LIN {X 0,Y 675.561,Z 368.02,A -85,B 0,C 180,E1 -4011.807,E2 -4011.807} C_VEL
LIN {X 0,Y 675.363,Z 376.661,A -85,B 0,C 180,E1 -4012.443,E2 -4012.443} C_VEL
LIN {X 0,Y 680.703,Z 399.355,A -85,B 0,C 180,E1 -4013.079,E2 -4013.079} C_VEL
LIN {X 0,Y 678.008,Z 663.117,A -85,B 0,C 180,E1 -4016.26,E2 -4016.26} C_VEL
LIN {X 0,Y 676.914,Z 767.818,A -85,B 0,C 180,E1 -4017.526,E2 -4017.526} C_VEL
LIN {X 0,Y 676.255,Z 793.274,A -85,B 0,C 180,E1 -4017.987,E2 -4017.987} C_VEL
LIN {X 0,Y 675.528,Z 814.444,A -85,B 0,C 180,E1 -4018.503,E2 -4018.503} C_VEL
LIN {X 0,Y 674.622,Z 838.547,A -85,B 0,C 180,E1 -4019.247,E2 -4019.247} C_VEL
LIN {X 0,Y 673.655,Z 859.342,A -85,B 0,C 180,E1 -4020.036,E2 -4020.036} C_VEL
LIN {X 0,Y 672.656,Z 880.17,A -85,B 0,C 180,E1 -4020.961,E2 -4020.961} C_VEL
LIN {X 0,Y 671.429,Z 902.313,A -85,B 0,C 180,E1 -4022.121,E2 -4022.121} C_VEL
LIN {X 0,Y 670.354,Z 922.188,A -85,B 0,C 180,E1 -4023.323,E2 -4023.323} C_VEL
LIN {X 0,Y 669.167,Z 942.614,A -85,B 0,C 180,E1 -4024.748,E2 -4024.748} C_VEL
LIN {X 0,Y 668.229,Z 959.683,A -85,B 0,C 180,E1 -4026.101,E2 -4026.101} C_VEL
LIN {X 0,Y 667.192,Z 978.606,A -85,B 0,C 180,E1 -4027.811,E2 -4027.811} C_VEL
LIN {X 0,Y 666.433,Z 993.633,A -85,B 0,C 180,E1 -4029.355,E2 -4029.355} C_VEL
LIN {X 0,Y 665.654,Z 1009.818,A -85,B 0,C 180,E1 -4031.249,E2 -4031.249} C_VEL
LIN {X 0,Y 665.145,Z 1022.539,A -85,B 0,C 180,E1 -4032.956,E2 -4032.956} C_VEL
LIN {X 0,Y 664.665,Z 1035.765,A -85,B 0,C 180,E1 -4035.004,E2 -4035.004} C_VEL
LIN {X 0,Y 664.369,Z 1045.92,A -85,B 0,C 180,E1 -4036.844,E2 -4036.844} C_VEL
LIN {X 0,Y 664.133,Z 1055.927,A -85,B 0,C 180,E1 -4039,E2 -4039} C_VEL
LIN {X 0,Y 664.022,Z 1062.817,A -85,B 0,C 180,E1 -4040.815,E2 -4040.815} C_VEL
LIN {X 0,Y 663.962,Z 1069.244,A -85,B 0,C 180,E1 -4042.907,E2 -4042.907} C_VEL
LIN {X 0,Y 663.925,Z 1073.656,A -85,B 0,C 180,E1 -4044.902,E2 -4044.902} C_VEL
LIN {X 0,Y 663.917,Z 1076.574,A -85,B 0,C 180,E1 -4046.806,E2 -4046.806} C_VEL
LIN {X 0,Y 663.91,Z 1078.261,A -85,B 0,C 180,E1 -4049.051,E2 -4049.051} C_VEL
LIN {X 0,Y 663.905,Z 1078.283,A -85,B 0,C 180,E1 -4050.863,E2 -4050.863} C_VEL
LIN {X 0,Y 663.916,Z 1076.799,A -85,B 0,C 180,E1 -4053.022,E2 -4053.022} C_VEL
LIN {X 0,Y 663.925,Z 1073.815,A -85,B 0,C 180,E1 -4055.011,E2 -4055.011} C_VEL
LIN {X 0,Y 663.956,Z 1069.451,A -85,B 0,C 180,E1 -4057.007,E2 -4057.007} C_VEL
LIN {X 0,Y 664.011,Z 1063.119,A -85,B 0,C 180,E1 -4059.097,E2 -4059.097} C_VEL
LIN {X 0,Y 664.128,Z 1056.186,A -85,B 0,C 180,E1 -4060.935,E2 -4060.935} C_VEL
LIN {X 0,Y 664.356,Z 1046.484,A -85,B 0,C 180,E1 -4063.047,E2 -4063.047} C_VEL
LIN {X 0,Y 664.649,Z 1036.288,A -85,B 0,C 180,E1 -4064.907,E2 -4064.907} C_VEL
LIN {X 0,Y 665.121,Z 1023.16,A -85,B 0,C 180,E1 -4066.956,E2 -4066.956} C_VEL
LIN {X 0,Y 665.624,Z 1010.525,A -85,B 0,C 180,E1 -4068.661,E2 -4068.661} C_VEL
LIN {X 0,Y 666.404,Z 994.378,A -85,B 0,C 180,E1 -4070.565,E2 -4070.565} C_VEL
LIN {X 0,Y 667.168,Z 979.013,A -85,B 0,C 180,E1 -4072.149,E2 -4072.149} C_VEL
LIN {X 0,Y 668.189,Z 960.506,A -85,B 0,C 180,E1 -4073.83,E2 -4073.83} C_VEL
LIN {X 0,Y 669.129,Z 943.22,A -85,B 0,C 180,E1 -4075.206,E2 -4075.206} C_VEL
LIN {X 0,Y 670.317,Z 922.909,A -85,B 0,C 180,E1 -4076.631,E2 -4076.631} C_VEL
LIN {X 0,Y 671.389,Z 903.048,A -85,B 0,C 180,E1 -4077.837,E2 -4077.837} C_VEL
LIN {X 0,Y 672.604,Z 881.268,A -85,B 0,C 180,E1 -4078.988,E2 -4078.988} C_VEL
LIN {X 0,Y 673.605,Z 860.476,A -85,B 0,C 180,E1 -4079.918,E2 -4079.918} C_VEL
LIN {X 0,Y 674.538,Z 840.351,A -85,B 0,C 180,E1 -4080.688,E2 -4080.688} C_VEL
LIN {X 0,Y 675.503,Z 815.099,A -85,B 0,C 180,E1 -4081.479,E2 -4081.479} C_VEL
LIN {X 0,Y 676.235,Z 793.801,A -85,B 0,C 180,E1 -4082.002,E2 -4082.002} C_VEL
LIN {X 0,Y 676.909,Z 768.357,A -85,B 0,C 180,E1 -4082.466,E2 -4082.466} C_VEL
LIN {X 0,Y 677.778,Z 687.025,A -85,B 0,C 180,E1 -4083.455,E2 -4083.455} C_VEL
LIN {X 0,Y 680.316,Z 433.987,A -85,B 0,C 180,E1 -4086.5,E2 -4086.5} C_VEL
LIN {X 0,Y 680.519,Z 397.746,A -85,B 0,C 180,E1 -4086.954,E2 -4086.954} C_VEL
LIN {X 0,Y 675.309,Z 375.991,A -85,B 0,C 180,E1 -4087.591,E2 -4087.591} C_VEL
LIN {X 0,Y 675.511,Z 367.275,A -85,B 0,C 180,E1 -4088.256,E2 -4088.256} C_VEL
LIN {X 0,Y 667.62,Z 346.692,A -85,B 0,C 180,E1 -4090.429,E2 -4090.429} C_VEL
LIN {X 0,Y 664.607,Z 338.449,A -85,B 0,C 180,E1 -4091.345,E2 -4091.345} C_VEL
LIN {X 0,Y 664.579,Z 338.447,A -85,B 0,C 180,E1 -4094.035,E2 -4094.035} C_VEL
LIN {X 0,Y 664.647,Z 338.444,A -85,B 0,C 180,E1 -4097.04,E2 -4097.04} C_VEL
LIN {X 0,Y 664.579,Z 338.439,A -85,B 0,C 180,E1 -4099.913,E2 -4099.913} C_VEL
LIN {X 0,Y 664.618,Z 338.438,A -85,B 0,C 180,E1 -4102.678,E2 -4102.678} C_VEL
LIN {X 0,Y 664.591,Z 338.44,A -85,B 0,C 180,E1 -4105.758,E2 -4105.758} C_VEL
LIN {X 0,Y 664.585,Z 338.439,A -85,B 0,C 180,E1 -4108.427,E2 -4108.427} C_VEL
LIN {X 0,Y 664.636,Z 338.439,A -85,B 0,C 180,E1 -4111.471,E2 -4111.471} C_VEL
LIN {X 0,Y 664.579,Z 338.441,A -85,B 0,C 180,E1 -4114.322,E2 -4114.322} C_VEL
LIN {X 0,Y 664.652,Z 338.43,A -85,B 0,C 180,E1 -4117.255,E2 -4117.255} C_VEL
LIN {X 0,Y 664.581,Z 338.436,A -85,B 0,C 180,E1 -4120.213,E2 -4120.213} C_VEL
LIN {X 0,Y 664.62,Z 338.438,A -85,B 0,C 180,E1 -4123.03,E2 -4123.03} C_VEL
LIN {X 0,Y 664.595,Z 338.44,A -85,B 0,C 180,E1 -4126.071,E2 -4126.071} C_VEL
LIN {X 0,Y 664.589,Z 338.44,A -85,B 0,C 180,E1 -4128.809,E2 -4128.809} C_VEL
LIN {X 0,Y 664.617,Z 338.445,A -85,B 0,C 180,E1 -4131.957,E2 -4131.957} C_VEL
LIN {X 0,Y 664.581,Z 338.436,A -85,B 0,C 180,E1 -4134.734,E2 -4134.734} C_VEL
LIN {X 0,Y 664.649,Z 338.44,A -85,B 0,C 180,E1 -4137.758,E2 -4137.758} C_VEL
LIN {X 0,Y 664.58,Z 338.43,A -85,B 0,C 180,E1 -4140.603,E2 -4140.603} C_VEL
LIN {X 0,Y 664.629,Z 338.438,A -85,B 0,C 180,E1 -4143.45,E2 -4143.45} C_VEL
LIN {X 0,Y 664.592,Z 338.438,A -85,B 0,C 180,E1 -4146.479,E2 -4146.479} C_VEL
LIN {X 0,Y 664.593,Z 338.44,A -85,B 0,C 180,E1 -4149.177,E2 -4149.177} C_VEL
LIN {X 0,Y 664.615,Z 338.443,A -85,B 0,C 180,E1 -4152.335,E2 -4152.335} C_VEL
LIN {X 0,Y 664.584,Z 338.437,A -85,B 0,C 180,E1 -4155.087,E2 -4155.087} C_VEL
LIN {X 0,Y 664.65,Z 338.438,A -85,B 0,C 180,E1 -4158.054,E2 -4158.054} C_VEL
LIN {X 0,Y 664.582,Z 338.434,A -85,B 0,C 180,E1 -4160.982,E2 -4160.982} C_VEL
LIN {X 0,Y 664.64,Z 338.439,A -85,B 0,C 180,E1 -4163.872,E2 -4163.872} C_VEL
LIN {X 0,Y 664.589,Z 338.443,A -85,B 0,C 180,E1 -4166.928,E2 -4166.928} C_VEL
LIN {X 0,Y 664.605,Z 338.431,A -85,B 0,C 180,E1 -4169.668,E2 -4169.668} C_VEL
LIN {X 0,Y 664.605,Z 338.436,A -85,B 0,C 180,E1 -4172.794,E2 -4172.794} C_VEL
LIN {X 0,Y 664.589,Z 338.441,A -85,B 0,C 180,E1 -4175.517,E2 -4175.517} C_VEL
LIN {X 0,Y 664.648,Z 338.437,A -85,B 0,C 180,E1 -4176.373,E2 -4176.373} C_VEL
LIN {X 0,Y 663.642,Z 338.561,A -85,B 0,C 180,E1 -4177.037,E2 -4177.037} C_VEL
LIN {X 0,Y 657.183,Z 339.369,A -85,B 0,C 180,E1 -4178.898,E2 -4178.898} C_VEL
LIN {X 0,Y 656.644,Z 339.428,A -85,B 0,C 180,E1 -4179.383,E2 -4179.383} C_VEL
LIN {X 0,Y 656.711,Z 339.428,A -85,B 0,C 180,E1 -4182.298,E2 -4182.298} C_VEL
LIN {X 0,Y 656.647,Z 339.421,A -85,B 0,C 180,E1 -4185.326,E2 -4185.326} C_VEL
LIN {X 0,Y 656.688,Z 339.425,A -85,B 0,C 180,E1 -4188.171,E2 -4188.171} C_VEL
LIN {X 0,Y 656.656,Z 339.438,A -85,B 0,C 180,E1 -4191.257,E2 -4191.257} C_VEL
LIN {X 0,Y 656.715,Z 339.481,A -85,B 0,C 180,E1 -4192.392,E2 -4192.392} C_VEL
LIN {X 0,Y 660.299,Z 349.162,A -85,B 0,C 180,E1 -4193.484,E2 -4193.484} C_VEL
LIN {X 0,Y 672.665,Z 370.1,A -85,B 0,C 180,E1 -4194.601,E2 -4194.601} C_VEL
LIN {X 0,Y 674.3,Z 373.32,A -85,B 0,C 180,E1 -4194.751,E2 -4194.751} C_VEL
LIN {X 0,Y 671.619,Z 610.249,A -85,B 0,C 180,E1 -4197.648,E2 -4197.648} C_VEL
LIN {X 0,Y 670.159,Z 737.628,A -85,B 0,C 180,E1 -4199.2,E2 -4199.2} C_VEL
LIN {X 0,Y 669.456,Z 763.152,A -85,B 0,C 180,E1 -4199.664,E2 -4199.664} C_VEL
LIN {X 0,Y 668.682,Z 784.147,A -85,B 0,C 180,E1 -4200.179,E2 -4200.179} C_VEL
LIN {X 0,Y 667.747,Z 806.973,A -85,B 0,C 180,E1 -4200.879,E2 -4200.879} C_VEL
LIN {X 0,Y 666.641,Z 828.781,A -85,B 0,C 180,E1 -4201.708,E2 -4201.708} C_VEL
LIN {X 0,Y 665.571,Z 849.482,A -85,B 0,C 180,E1 -4202.632,E2 -4202.632} C_VEL
LIN {X 0,Y 664.202,Z 872.164,A -85,B 0,C 180,E1 -4203.827,E2 -4203.827} C_VEL
LIN {X 0,Y 663.039,Z 891.79,A -85,B 0,C 180,E1 -4205.023,E2 -4205.023} C_VEL
LIN {X 0,Y 661.729,Z 912.624,A -85,B 0,C 180,E1 -4206.49,E2 -4206.49} C_VEL
LIN {X 0,Y 660.649,Z 930.299,A -85,B 0,C 180,E1 -4207.907,E2 -4207.907} C_VEL
LIN {X 0,Y 659.548,Z 948.684,A -85,B 0,C 180,E1 -4209.593,E2 -4209.593} C_VEL
LIN {X 0,Y 658.704,Z 963.538,A -85,B 0,C 180,E1 -4211.136,E2 -4211.136} C_VEL
LIN {X 0,Y 657.869,Z 979.584,A -85,B 0,C 180,E1 -4213.033,E2 -4213.033} C_VEL
LIN {X 0,Y 657.3,Z 992.193,A -85,B 0,C 180,E1 -4214.742,E2 -4214.742} C_VEL
LIN {X 0,Y 656.765,Z 1005.394,A -85,B 0,C 180,E1 -4216.799,E2 -4216.799} C_VEL
LIN {X 0,Y 656.44,Z 1015.162,A -85,B 0,C 180,E1 -4218.579,E2 -4218.579} C_VEL
LIN {X 0,Y 656.198,Z 1024.753,A -85,B 0,C 180,E1 -4220.616,E2 -4220.616} C_VEL
LIN {X 0,Y 656.045,Z 1032.462,A -85,B 0,C 180,E1 -4222.644,E2 -4222.644} C_VEL
LIN {X 0,Y 655.954,Z 1038.693,A -85,B 0,C 180,E1 -4224.665,E2 -4224.665} C_VEL
LIN {X 0,Y 655.916,Z 1043.44,A -85,B 0,C 180,E1 -4226.767,E2 -4226.767} C_VEL
LIN {X 0,Y 655.912,Z 1046.306,A -85,B 0,C 180,E1 -4228.602,E2 -4228.602} C_VEL
LIN {X 0,Y 655.909,Z 1048.183,A -85,B 0,C 180,E1 -4230.786,E2 -4230.786} C_VEL
LIN {X 0,Y 655.896,Z 1048.337,A -85,B 0,C 180,E1 -4232.709,E2 -4232.709} C_VEL
LIN {X 0,Y 655.897,Z 1047.251,A -85,B 0,C 180,E1 -4234.634,E2 -4234.634} C_VEL
LIN {X 0,Y 655.914,Z 1044.339,A -85,B 0,C 180,E1 -4236.829,E2 -4236.829} C_VEL
LIN {X 0,Y 655.935,Z 1040.525,A -85,B 0,C 180,E1 -4238.68,E2 -4238.68} C_VEL
LIN {X 0,Y 655.991,Z 1034.958,A -85,B 0,C 180,E1 -4240.717,E2 -4240.717} C_VEL
LIN {X 0,Y 656.126,Z 1027.58,A -85,B 0,C 180,E1 -4242.766,E2 -4242.766} C_VEL
LIN {X 0,Y 656.332,Z 1019.332,A -85,B 0,C 180,E1 -4244.671,E2 -4244.671} C_VEL
LIN {X 0,Y 656.66,Z 1008.638,A -85,B 0,C 180,E1 -4246.726,E2 -4246.726} C_VEL
LIN {X 0,Y 657.063,Z 997.584,A -85,B 0,C 180,E1 -4248.547,E2 -4248.547} C_VEL
LIN {X 0,Y 657.693,Z 983.412,A -85,B 0,C 180,E1 -4250.56,E2 -4250.56} C_VEL
LIN {X 0,Y 658.362,Z 970.013,A -85,B 0,C 180,E1 -4252.22,E2 -4252.22} C_VEL
LIN {X 0,Y 659.305,Z 952.896,A -85,B 0,C 180,E1 -4254.078,E2 -4254.078} C_VEL
LIN {X 0,Y 660.218,Z 937.24,A -85,B 0,C 180,E1 -4255.571,E2 -4255.571} C_VEL
LIN {X 0,Y 661.416,Z 917.701,A -85,B 0,C 180,E1 -4257.213,E2 -4257.213} C_VEL
LIN {X 0,Y 662.557,Z 899.324,A -85,B 0,C 180,E1 -4258.559,E2 -4258.559} C_VEL
LIN {X 0,Y 663.909,Z 877.57,A -85,B 0,C 180,E1 -4259.951,E2 -4259.951} C_VEL
LIN {X 0,Y 665.051,Z 857.744,A -85,B 0,C 180,E1 -4261.044,E2 -4261.044} C_VEL
LIN {X 0,Y 666.366,Z 834.681,A -85,B 0,C 180,E1 -4262.136,E2 -4262.136} C_VEL
LIN {X 0,Y 667.387,Z 814.243,A -85,B 0,C 180,E1 -4262.946,E2 -4262.946} C_VEL
LIN {X 0,Y 668.356,Z 792.889,A -85,B 0,C 180,E1 -4263.661,E2 -4263.661} C_VEL
LIN {X 0,Y 669.253,Z 768.222,A -85,B 0,C 180,E1 -4264.313,E2 -4264.313} C_VEL
LIN {X 0,Y 669.946,Z 746.408,A -85,B 0,C 180,E1 -4264.75,E2 -4264.75} C_VEL
LIN {X 0,Y 670.503,Z 714.244,A -85,B 0,C 180,E1 -4265.192,E2 -4265.192} C_VEL
LIN {X 0,Y 673.317,Z 459.697,A -85,B 0,C 180,E1 -4268.273,E2 -4268.273} C_VEL
LIN {X 0,Y 674.117,Z 372.503,A -85,B 0,C 180,E1 -4269.362,E2 -4269.362} C_VEL
LIN {X 0,Y 662.206,Z 352.425,A -85,B 0,C 180,E1 -4270.43,E2 -4270.43} C_VEL
LIN {X 0,Y 659.951,Z 348.526,A -85,B 0,C 180,E1 -4270.654,E2 -4270.654} C_VEL
LIN {X 0,Y 656.699,Z 339.432,A -85,B 0,C 180,E1 -4271.748,E2 -4271.748} C_VEL
LIN {X 0,Y 656.644,Z 339.431,A -85,B 0,C 180,E1 -4274.586,E2 -4274.586} C_VEL
LIN {X 0,Y 656.713,Z 339.426,A -85,B 0,C 180,E1 -4277.585,E2 -4277.585} C_VEL
LIN {X 0,Y 656.644,Z 339.425,A -85,B 0,C 180,E1 -4280.536,E2 -4280.536} C_VEL
LIN {X 0,Y 656.686,Z 339.413,A -85,B 0,C 180,E1 -4283.362,E2 -4283.362} C_VEL
LIN {X 0,Y 656.653,Z 339.43,A -85,B 0,C 180,E1 -4286.444,E2 -4286.444} C_VEL
LIN {X 0,Y 656.662,Z 339.428,A -85,B 0,C 180,E1 -4289.228,E2 -4289.228} C_VEL
LIN {X 0,Y 656.661,Z 339.429,A -85,B 0,C 180,E1 -4292.426,E2 -4292.426} C_VEL
LIN {X 0,Y 656.65,Z 339.426,A -85,B 0,C 180,E1 -4295.167,E2 -4295.167} C_VEL
LIN {X 0,Y 656.688,Z 339.422,A -85,B 0,C 180,E1 -4298.284,E2 -4298.284} C_VEL
LIN {X 0,Y 656.643,Z 339.431,A -85,B 0,C 180,E1 -4301.074,E2 -4301.074} C_VEL
LIN {X 0,Y 656.712,Z 339.428,A -85,B 0,C 180,E1 -4304.094,E2 -4304.094} C_VEL
LIN {X 0,Y 656.642,Z 339.428,A -85,B 0,C 180,E1 -4307.045,E2 -4307.045} C_VEL
LIN {X 0,Y 656.706,Z 339.423,A -85,B 0,C 180,E1 -4310.004,E2 -4310.004} C_VEL
LIN {X 0,Y 656.646,Z 339.429,A -85,B 0,C 180,E1 -4313.003,E2 -4313.003} C_VEL
LIN {X 0,Y 656.675,Z 339.429,A -85,B 0,C 180,E1 -4315.819,E2 -4315.819} C_VEL
LIN {X 0,Y 656.652,Z 339.423,A -85,B 0,C 180,E1 -4318.953,E2 -4318.953} C_VEL
LIN {X 0,Y 656.651,Z 339.433,A -85,B 0,C 180,E1 -4321.658,E2 -4321.658} C_VEL
LIN {X 0,Y 656.676,Z 339.428,A -85,B 0,C 180,E1 -4324.804,E2 -4324.804} C_VEL
LIN {X 0,Y 656.642,Z 339.423,A -85,B 0,C 180,E1 -4327.613,E2 -4327.613} C_VEL
LIN {X 0,Y 656.706,Z 339.419,A -85,B 0,C 180,E1 -4330.616,E2 -4330.616} C_VEL
LIN {X 0,Y 656.64,Z 339.431,A -85,B 0,C 180,E1 -4333.562,E2 -4333.562} C_VEL
LIN {X 0,Y 656.707,Z 339.425,A -85,B 0,C 180,E1 -4336.451,E2 -4336.451} C_VEL
LIN {X 0,Y 656.641,Z 339.421,A -85,B 0,C 180,E1 -4339.48,E2 -4339.48} C_VEL
LIN {X 0,Y 656.676,Z 339.434,A -85,B 0,C 180,E1 -4342.281,E2 -4342.281} C_VEL
LIN {X 0,Y 656.65,Z 339.43,A -85,B 0,C 180,E1 -4345.43,E2 -4345.43} C_VEL
LIN {X 0,Y 656.655,Z 339.429,A -85,B 0,C 180,E1 -4348.167,E2 -4348.167} C_VEL
LIN {X 0,Y 656.659,Z 339.43,A -85,B 0,C 180,E1 -4351.383,E2 -4351.383} C_VEL
LIN {X 0,Y 656.643,Z 339.434,A -85,B 0,C 180,E1 -4354.081,E2 -4354.081} C_VEL
LIN {X 0,Y 656.707,Z 339.429,A -85,B 0,C 180,E1 -4357.081,E2 -4357.081} C_VEL
LIN {X 0,Y 656.639,Z 339.434,A -85,B 0,C 180,E1 -4359.986,E2 -4359.986} C_VEL
LIN {X 0,Y 656.706,Z 339.421,A -85,B 0,C 180,E1 -4362.915,E2 -4362.915} C_VEL
LIN {X 0,Y 656.641,Z 339.434,A -85,B 0,C 180,E1 -4365.95,E2 -4365.95} C_VEL
LIN {X 0,Y 656.657,Z 339.564,A -85,B 0,C 180,E1 -4368.169,E2 -4368.169} C_VEL
LIN {X 0,Y 665.444,Z 362.462,A -85,B 0,C 180,E1 -4370.7,E2 -4370.7} C_VEL
LIN {X 0,Y 668.552,Z 371.163,A -85,B 0,C 180,E1 -4371.601,E2 -4371.601} C_VEL
LIN {X 0,Y 668.496,Z 376.599,A -85,B 0,C 180,E1 -4371.992,E2 -4371.992} C_VEL
LIN {X 0,Y 674.269,Z 401.065,A -85,B 0,C 180,E1 -4372.692,E2 -4372.692} C_VEL
LIN {X 0,Y 671.314,Z 665.842,A -85,B 0,C 180,E1 -4375.914,E2 -4375.914} C_VEL
LIN {X 0,Y 670.159,Z 767.71,A -85,B 0,C 180,E1 -4377.156,E2 -4377.156} C_VEL
LIN {X 0,Y 669.461,Z 793.012,A -85,B 0,C 180,E1 -4377.616,E2 -4377.616} C_VEL
LIN {X 0,Y 668.687,Z 814.008,A -85,B 0,C 180,E1 -4378.131,E2 -4378.131} C_VEL
LIN {X 0,Y 667.732,Z 837.259,A -85,B 0,C 180,E1 -4378.844,E2 -4378.844} C_VEL
LIN {X 0,Y 666.67,Z 858.208,A -85,B 0,C 180,E1 -4379.639,E2 -4379.639} C_VEL
LIN {X 0,Y 665.63,Z 878.27,A -85,B 0,C 180,E1 -4380.53,E2 -4380.53} C_VEL
LIN {X 0,Y 664.254,Z 901.417,A -85,B 0,C 180,E1 -4381.739,E2 -4381.739} C_VEL
LIN {X 0,Y 663.095,Z 920.728,A -85,B 0,C 180,E1 -4382.91,E2 -4382.91} C_VEL
LIN {X 0,Y 661.775,Z 942.003,A -85,B 0,C 180,E1 -4384.398,E2 -4384.398} C_VEL
LIN {X 0,Y 660.695,Z 959.4,A -85,B 0,C 180,E1 -4385.787,E2 -4385.787} C_VEL
LIN {X 0,Y 659.552,Z 978.604,A -85,B 0,C 180,E1 -4387.54,E2 -4387.54} C_VEL
LIN {X 0,Y 658.706,Z 993.631,A -85,B 0,C 180,E1 -4389.101,E2 -4389.101} C_VEL
LIN {X 0,Y 657.857,Z 1009.82,A -85,B 0,C 180,E1 -4391.018,E2 -4391.018} C_VEL
LIN {X 0,Y 657.284,Z 1022.521,A -85,B 0,C 180,E1 -4392.744,E2 -4392.744} C_VEL
LIN {X 0,Y 656.745,Z 1035.972,A -85,B 0,C 180,E1 -4394.855,E2 -4394.855} C_VEL
LIN {X 0,Y 656.42,Z 1046.022,A -85,B 0,C 180,E1 -4396.702,E2 -4396.702} C_VEL
LIN {X 0,Y 656.155,Z 1056.164,A -85,B 0,C 180,E1 -4398.924,E2 -4398.924} C_VEL
LIN {X 0,Y 656.032,Z 1063.12,A -85,B 0,C 180,E1 -4400.791,E2 -4400.791} C_VEL
LIN {X 0,Y 655.964,Z 1069.45,A -85,B 0,C 180,E1 -4402.908,E2 -4402.908} C_VEL
LIN {X 0,Y 655.926,Z 1073.816,A -85,B 0,C 180,E1 -4404.928,E2 -4404.928} C_VEL
LIN {X 0,Y 655.917,Z 1076.8,A -85,B 0,C 180,E1 -4406.942,E2 -4406.942} C_VEL
LIN {X 0,Y 655.906,Z 1078.283,A -85,B 0,C 180,E1 -4409.127,E2 -4409.127} C_VEL
LIN {X 0,Y 655.91,Z 1078.26,A -85,B 0,C 180,E1 -4410.961,E2 -4410.961} C_VEL
LIN {X 0,Y 655.917,Z 1076.574,A -85,B 0,C 180,E1 -4413.233,E2 -4413.233} C_VEL
LIN {X 0,Y 655.925,Z 1073.655,A -85,B 0,C 180,E1 -4415.16,E2 -4415.16} C_VEL
LIN {X 0,Y 655.96,Z 1069.016,A -85,B 0,C 180,E1 -4417.268,E2 -4417.268} C_VEL
LIN {X 0,Y 656.041,Z 1062.816,A -85,B 0,C 180,E1 -4419.297,E2 -4419.297} C_VEL
LIN {X 0,Y 656.163,Z 1055.832,A -85,B 0,C 180,E1 -4421.159,E2 -4421.159} C_VEL
LIN {X 0,Y 656.42,Z 1046.025,A -85,B 0,C 180,E1 -4423.298,E2 -4423.298} C_VEL
LIN {X 0,Y 656.745,Z 1035.974,A -85,B 0,C 180,E1 -4425.145,E2 -4425.145} C_VEL
LIN {X 0,Y 657.284,Z 1022.523,A -85,B 0,C 180,E1 -4427.256,E2 -4427.256} C_VEL
LIN {X 0,Y 657.857,Z 1009.82,A -85,B 0,C 180,E1 -4428.981,E2 -4428.981} C_VEL
LIN {X 0,Y 658.706,Z 993.631,A -85,B 0,C 180,E1 -4430.899,E2 -4430.899} C_VEL
LIN {X 0,Y 659.552,Z 978.605,A -85,B 0,C 180,E1 -4432.46,E2 -4432.46} C_VEL
LIN {X 0,Y 660.724,Z 958.846,A -85,B 0,C 180,E1 -4434.259,E2 -4434.259} C_VEL
LIN {X 0,Y 661.83,Z 941.235,A -85,B 0,C 180,E1 -4435.66,E2 -4435.66} C_VEL
LIN {X 0,Y 663.131,Z 919.985,A -85,B 0,C 180,E1 -4437.137,E2 -4437.137} C_VEL
LIN {X 0,Y 664.304,Z 900.683,A -85,B 0,C 180,E1 -4438.303,E2 -4438.303} C_VEL
LIN {X 0,Y 665.679,Z 877.27,A -85,B 0,C 180,E1 -4439.517,E2 -4439.517} C_VEL
LIN {X 0,Y 666.708,Z 857.462,A -85,B 0,C 180,E1 -4440.392,E2 -4440.392} C_VEL
LIN {X 0,Y 667.886,Z 833.797,A -85,B 0,C 180,E1 -4441.271,E2 -4441.271} C_VEL
LIN {X 0,Y 668.755,Z 812.386,A -85,B 0,C 180,E1 -4441.913,E2 -4441.913} C_VEL
LIN {X 0,Y 669.581,Z 790.077,A -85,B 0,C 180,E1 -4442.449,E2 -4442.449} C_VEL
LIN {X 0,Y 670.189,Z 765.252,A -85,B 0,C 180,E1 -4442.879,E2 -4442.879} C_VEL
LIN {X 0,Y 672.804,Z 526.404,A -85,B 0,C 180,E1 -4445.774,E2 -4445.774} C_VEL
LIN {X 0,Y 674.093,Z 399.551,A -85,B 0,C 180,E1 -4447.339,E2 -4447.339} C_VEL
LIN {X 0,Y 668.399,Z 375.76,A -85,B 0,C 180,E1 -4448.049,E2 -4448.049} C_VEL
LIN {X 0,Y 668.438,Z 370.567,A -85,B 0,C 180,E1 -4448.456,E2 -4448.456} C_VEL
LIN {X 0,Y 660.208,Z 348.828,A -85,B 0,C 180,E1 -4450.777,E2 -4450.777} C_VEL
LIN {X 0,Y 656.64,Z 339.439,A -85,B 0,C 180,E1 -4451.833,E2 -4451.833} C_VEL
LIN {X 0,Y 656.699,Z 339.433,A -85,B 0,C 180,E1 -4454.704,E2 -4454.704} C_VEL
LIN {X 0,Y 656.645,Z 339.436,A -85,B 0,C 180,E1 -4457.735,E2 -4457.735} C_VEL
LIN {X 0,Y 656.66,Z 339.425,A -85,B 0,C 180,E1 -4460.47,E2 -4460.47} C_VEL
LIN {X 0,Y 656.656,Z 339.435,A -85,B 0,C 180,E1 -4463.677,E2 -4463.677} C_VEL
LIN {X 0,Y 656.648,Z 339.427,A -85,B 0,C 180,E1 -4466.401,E2 -4466.401} C_VEL
LIN {X 0,Y 656.683,Z 339.427,A -85,B 0,C 180,E1 -4469.533,E2 -4469.533} C_VEL
LIN {X 0,Y 656.642,Z 339.423,A -85,B 0,C 180,E1 -4472.326,E2 -4472.326} C_VEL
LIN {X 0,Y 656.711,Z 339.428,A -85,B 0,C 180,E1 -4475.364,E2 -4475.364} C_VEL
LIN {X 0,Y 656.639,Z 339.431,A -85,B 0,C 180,E1 -4478.283,E2 -4478.283} C_VEL
LIN {X 0,Y 656.699,Z 339.419,A -85,B 0,C 180,E1 -4481.168,E2 -4481.168} C_VEL
LIN {X 0,Y 656.646,Z 339.428,A -85,B 0,C 180,E1 -4484.23,E2 -4484.23} C_VEL
LIN {X 0,Y 656.673,Z 339.424,A -85,B 0,C 180,E1 -4487.034,E2 -4487.034} C_VEL
LIN {X 0,Y 656.653,Z 339.421,A -85,B 0,C 180,E1 -4490.181,E2 -4490.181} C_VEL
LIN {X 0,Y 656.653,Z 339.429,A -85,B 0,C 180,E1 -4492.915,E2 -4492.915} C_VEL
LIN {X 0,Y 656.673,Z 339.425,A -85,B 0,C 180,E1 -4496.071,E2 -4496.071} C_VEL
LIN {X 0,Y 656.646,Z 339.429,A -85,B 0,C 180,E1 -4498.866,E2 -4498.866} C_VEL
LIN {X 0,Y 656.702,Z 339.423,A -85,B 0,C 180,E1 -4501.92,E2 -4501.92} C_VEL
LIN {X 0,Y 656.642,Z 339.426,A -85,B 0,C 180,E1 -4504.804,E2 -4504.804} C_VEL
LIN {X 0,Y 656.712,Z 339.424,A -85,B 0,C 180,E1 -4507.788,E2 -4507.788} C_VEL
LIN {X 0,Y 656.642,Z 339.419,A -85,B 0,C 180,E1 -4510.795,E2 -4510.795} C_VEL
LIN {X 0,Y 656.704,Z 339.427,A -85,B 0,C 180,E1 -4513.733,E2 -4513.733} C_VEL
LIN {X 0,Y 656.649,Z 339.428,A -85,B 0,C 180,E1 -4516.726,E2 -4516.726} C_VEL
LIN {X 0,Y 656.668,Z 339.428,A -85,B 0,C 180,E1 -4519.519,E2 -4519.519} C_VEL
LIN {X 0,Y 656.662,Z 339.433,A -85,B 0,C 180,E1 -4522.669,E2 -4522.669} C_VEL
LIN {X 0,Y 656.65,Z 339.419,A -85,B 0,C 180,E1 -4525.43,E2 -4525.43} C_VEL
LIN {X 0,Y 656.683,Z 339.425,A -85,B 0,C 180,E1 -4528.562,E2 -4528.562} C_VEL
LIN {X 0,Y 656.647,Z 339.431,A -85,B 0,C 180,E1 -4531.384,E2 -4531.384} C_VEL
LIN {X 0,Y 656.708,Z 339.425,A -85,B 0,C 180,E1 -4534.394,E2 -4534.394} C_VEL
LIN {X 0,Y 656.645,Z 339.43,A -85,B 0,C 180,E1 -4537.358,E2 -4537.358} C_VEL
LIN {X 0,Y 656.644,Z 339.428,A -85,B 0,C 180,E1 -4539.383,E2 -4539.383} C_VEL
LIN {X 0,Y 655.666,Z 339.552,A -85,B 0,C 180,E1 -4540.054,E2 -4540.054} C_VEL
LIN {X 0,Y 649.315,Z 340.354,A -85,B 0,C 180,E1 -4541.939,E2 -4541.939} C_VEL
LIN {X 0,Y 648.773,Z 340.412,A -85,B 0,C 180,E1 -4542.429,E2 -4542.429} C_VEL
LIN {X 0,Y 648.706,Z 340.41,A -85,B 0,C 180,E1 -4545.407,E2 -4545.407} C_VEL
LIN {X 0,Y 648.771,Z 340.413,A -85,B 0,C 180,E1 -4548.374,E2 -4548.374} C_VEL
LIN {X 0,Y 648.711,Z 340.428,A -85,B 0,C 180,E1 -4551.395,E2 -4551.395} C_VEL
LIN {X 0,Y 648.725,Z 340.49,A -85,B 0,C 180,E1 -4551.881,E2 -4551.881} C_VEL
LIN {X 0,Y 652.031,Z 349.362,A -85,B 0,C 180,E1 -4552.903,E2 -4552.903} C_VEL
LIN {X 0,Y 664.392,Z 369.862,A -85,B 0,C 180,E1 -4554.046,E2 -4554.046} C_VEL
LIN {X 0,Y 667.91,Z 376.435,A -85,B 0,C 180,E1 -4554.371,E2 -4554.371} C_VEL
LIN {X 0,Y 664.987,Z 613.857,A -85,B 0,C 180,E1 -4557.3,E2 -4557.3} C_VEL
LIN {X 0,Y 663.442,Z 737.836,A -85,B 0,C 180,E1 -4558.825,E2 -4558.825} C_VEL
LIN {X 0,Y 662.693,Z 763.181,A -85,B 0,C 180,E1 -4559.291,E2 -4559.291} C_VEL
LIN {X 0,Y 661.868,Z 783.905,A -85,B 0,C 180,E1 -4559.803,E2 -4559.803} C_VEL
LIN {X 0,Y 660.864,Z 806.43,A -85,B 0,C 180,E1 -4560.496,E2 -4560.496} C_VEL
LIN {X 0,Y 659.611,Z 829.135,A -85,B 0,C 180,E1 -4561.366,E2 -4561.366} C_VEL
LIN {X 0,Y 658.444,Z 850.054,A -85,B 0,C 180,E1 -4562.31,E2 -4562.31} C_VEL
LIN {X 0,Y 656.995,Z 872.245,A -85,B 0,C 180,E1 -4563.494,E2 -4563.494} C_VEL
LIN {X 0,Y 655.751,Z 891.2,A -85,B 0,C 180,E1 -4564.659,E2 -4564.659} C_VEL
LIN {X 0,Y 654.372,Z 911.773,A -85,B 0,C 180,E1 -4566.114,E2 -4566.114} C_VEL
LIN {X 0,Y 653.2,Z 928.979,A -85,B 0,C 180,E1 -4567.5,E2 -4567.5} C_VEL
LIN {X 0,Y 651.965,Z 948.038,A -85,B 0,C 180,E1 -4569.251,E2 -4569.251} C_VEL
LIN {X 0,Y 651.012,Z 963.172,A -85,B 0,C 180,E1 -4570.836,E2 -4570.836} C_VEL
LIN {X 0,Y 650.073,Z 979.79,A -85,B 0,C 180,E1 -4572.823,E2 -4572.823} C_VEL
LIN {X 0,Y 649.433,Z 992.376,A -85,B 0,C 180,E1 -4574.552,E2 -4574.552} C_VEL
LIN {X 0,Y 648.851,Z 1005.546,A -85,B 0,C 180,E1 -4576.635,E2 -4576.635} C_VEL
LIN {X 0,Y 648.499,Z 1015.294,A -85,B 0,C 180,E1 -4578.437,E2 -4578.437} C_VEL
LIN {X 0,Y 648.228,Z 1024.856,A -85,B 0,C 180,E1 -4580.5,E2 -4580.5} C_VEL
LIN {X 0,Y 648.057,Z 1032.549,A -85,B 0,C 180,E1 -4582.553,E2 -4582.553} C_VEL
LIN {X 0,Y 647.956,Z 1038.766,A -85,B 0,C 180,E1 -4584.599,E2 -4584.599} C_VEL
LIN {X 0,Y 647.917,Z 1043.485,A -85,B 0,C 180,E1 -4586.727,E2 -4586.727} C_VEL
LIN {X 0,Y 647.912,Z 1046.338,A -85,B 0,C 180,E1 -4588.585,E2 -4588.585} C_VEL
LIN {X 0,Y 647.909,Z 1048.189,A -85,B 0,C 180,E1 -4590.796,E2 -4590.796} C_VEL
LIN {X 0,Y 647.897,Z 1048.331,A -85,B 0,C 180,E1 -4592.742,E2 -4592.742} C_VEL
LIN {X 0,Y 647.897,Z 1047.231,A -85,B 0,C 180,E1 -4594.692,E2 -4594.692} C_VEL
LIN {X 0,Y 647.916,Z 1044.293,A -85,B 0,C 180,E1 -4596.914,E2 -4596.914} C_VEL
LIN {X 0,Y 647.938,Z 1040.673,A -85,B 0,C 180,E1 -4598.698,E2 -4598.698} C_VEL
LIN {X 0,Y 647.999,Z 1035.15,A -85,B 0,C 180,E1 -4600.761,E2 -4600.761} C_VEL
LIN {X 0,Y 648.144,Z 1027.81,A -85,B 0,C 180,E1 -4602.841,E2 -4602.841} C_VEL
LIN {X 0,Y 648.366,Z 1019.725,A -85,B 0,C 180,E1 -4604.741,E2 -4604.741} C_VEL
LIN {X 0,Y 648.748,Z 1008.485,A -85,B 0,C 180,E1 -4606.936,E2 -4606.936} C_VEL
LIN {X 0,Y 649.199,Z 997.43,A -85,B 0,C 180,E1 -4608.778,E2 -4608.778} C_VEL
LIN {X 0,Y 649.881,Z 983.201,A -85,B 0,C 180,E1 -4610.819,E2 -4610.819} C_VEL
LIN {X 0,Y 650.668,Z 969.379,A -85,B 0,C 180,E1 -4612.546,E2 -4612.546} C_VEL
LIN {X 0,Y 651.687,Z 952.296,A -85,B 0,C 180,E1 -4614.411,E2 -4614.411} C_VEL
LIN {X 0,Y 652.723,Z 936.319,A -85,B 0,C 180,E1 -4615.945,E2 -4615.945} C_VEL
LIN {X 0,Y 654.057,Z 916.102,A -85,B 0,C 180,E1 -4617.644,E2 -4617.644} C_VEL
LIN {X 0,Y 655.311,Z 897.949,A -85,B 0,C 180,E1 -4618.976,E2 -4618.976} C_VEL
LIN {X 0,Y 656.737,Z 876.257,A -85,B 0,C 180,E1 -4620.363,E2 -4620.363} C_VEL
LIN {X 0,Y 657.95,Z 857.206,A -85,B 0,C 180,E1 -4621.417,E2 -4621.417} C_VEL
LIN {X 0,Y 659.382,Z 833.782,A -85,B 0,C 180,E1 -4622.528,E2 -4622.528} C_VEL
LIN {X 0,Y 660.484,Z 813.484,A -85,B 0,C 180,E1 -4623.335,E2 -4623.335} C_VEL
LIN {X 0,Y 661.599,Z 790.536,A -85,B 0,C 180,E1 -4624.104,E2 -4624.104} C_VEL
LIN {X 0,Y 662.533,Z 766.989,A -85,B 0,C 180,E1 -4624.714,E2 -4624.714} C_VEL
LIN {X 0,Y 663.294,Z 744.574,A -85,B 0,C 180,E1 -4625.159,E2 -4625.159} C_VEL
LIN {X 0,Y 663.855,Z 710.877,A -85,B 0,C 180,E1 -4625.613,E2 -4625.613} C_VEL
LIN {X 0,Y 666.919,Z 456.369,A -85,B 0,C 180,E1 -4628.724,E2 -4628.724} C_VEL
LIN {X 0,Y 667.73,Z 375.714,A -85,B 0,C 180,E1 -4629.741,E2 -4629.741} C_VEL
LIN {X 0,Y 657.19,Z 357.792,A -85,B 0,C 180,E1 -4630.705,E2 -4630.705} C_VEL
LIN {X 0,Y 651.704,Z 348.634,A -85,B 0,C 180,E1 -4631.254,E2 -4631.254} C_VEL
LIN {X 0,Y 648.713,Z 340.425,A -85,B 0,C 180,E1 -4632.253,E2 -4632.253} C_VEL
LIN {X 0,Y 648.736,Z 340.421,A -85,B 0,C 180,E1 -4635.097,E2 -4635.097} C_VEL
LIN {X 0,Y 648.717,Z 340.413,A -85,B 0,C 180,E1 -4638.252,E2 -4638.252} C_VEL
LIN {X 0,Y 648.719,Z 340.416,A -85,B 0,C 180,E1 -4641.033,E2 -4641.033} C_VEL
LIN {X 0,Y 648.722,Z 340.393,A -85,B 0,C 180,E1 -4644.256,E2 -4644.256} C_VEL
LIN {X 0,Y 648.713,Z 340.422,A -85,B 0,C 180,E1 -4647.037,E2 -4647.037} C_VEL
LIN {X 0,Y 648.744,Z 340.417,A -85,B 0,C 180,E1 -4650.196,E2 -4650.196} C_VEL
LIN {X 0,Y 648.707,Z 340.421,A -85,B 0,C 180,E1 -4652.987,E2 -4652.987} C_VEL
LIN {X 0,Y 648.768,Z 340.418,A -85,B 0,C 180,E1 -4656.055,E2 -4656.055} C_VEL
LIN {X 0,Y 648.704,Z 340.414,A -85,B 0,C 180,E1 -4658.953,E2 -4658.953} C_VEL
LIN {X 0,Y 648.767,Z 340.412,A -85,B 0,C 180,E1 -4661.861,E2 -4661.861} C_VEL
LIN {X 0,Y 648.705,Z 340.418,A -85,B 0,C 180,E1 -4664.901,E2 -4664.901} C_VEL
LIN {X 0,Y 648.743,Z 340.42,A -85,B 0,C 180,E1 -4667.733,E2 -4667.733} C_VEL
LIN {X 0,Y 648.711,Z 340.415,A -85,B 0,C 180,E1 -4670.865,E2 -4670.865} C_VEL
LIN {X 0,Y 648.722,Z 340.421,A -85,B 0,C 180,E1 -4673.628,E2 -4673.628} C_VEL
LIN {X 0,Y 648.722,Z 340.418,A -85,B 0,C 180,E1 -4676.819,E2 -4676.819} C_VEL
LIN {X 0,Y 648.709,Z 340.415,A -85,B 0,C 180,E1 -4679.558,E2 -4679.558} C_VEL
LIN {X 0,Y 648.751,Z 340.408,A -85,B 0,C 180,E1 -4682.65,E2 -4682.65} C_VEL
LIN {X 0,Y 648.703,Z 340.421,A -85,B 0,C 180,E1 -4685.484,E2 -4685.484} C_VEL
LIN {X 0,Y 648.776,Z 340.417,A -85,B 0,C 180,E1 -4688.419,E2 -4688.419} C_VEL
LIN {X 0,Y 648.703,Z 340.409,A -85,B 0,C 180,E1 -4691.389,E2 -4691.389} C_VEL
LIN {X 0,Y 648.757,Z 340.418,A -85,B 0,C 180,E1 -4694.276,E2 -4694.276} C_VEL
LIN {X 0,Y 648.712,Z 340.418,A -85,B 0,C 180,E1 -4697.306,E2 -4697.306} C_VEL
LIN {X 0,Y 648.722,Z 340.412,A -85,B 0,C 180,E1 -4700.104,E2 -4700.104} C_VEL
LIN {X 0,Y 648.715,Z 340.41,A -85,B 0,C 180,E1 -4703.336,E2 -4703.336} C_VEL
LIN {X 0,Y 648.712,Z 340.422,A -85,B 0,C 180,E1 -4706.058,E2 -4706.058} C_VEL
LIN {X 0,Y 648.733,Z 340.417,A -85,B 0,C 180,E1 -4709.248,E2 -4709.248} C_VEL
LIN {X 0,Y 648.705,Z 340.422,A -85,B 0,C 180,E1 -4712.032,E2 -4712.032} C_VEL
LIN {X 0,Y 648.762,Z 340.42,A -85,B 0,C 180,E1 -4715.091,E2 -4715.091} C_VEL
LIN {X 0,Y 648.7,Z 340.421,A -85,B 0,C 180,E1 -4717.953,E2 -4717.953} C_VEL
LIN {X 0,Y 648.775,Z 340.418,A -85,B 0,C 180,E1 -4720.921,E2 -4720.921} C_VEL
LIN {X 0,Y 648.702,Z 340.422,A -85,B 0,C 180,E1 -4723.96,E2 -4723.96} C_VEL
LIN {X 0,Y 648.75,Z 340.417,A -85,B 0,C 180,E1 -4726.818,E2 -4726.818} C_VEL
LIN {X 0,Y 648.729,Z 340.449,A -85,B 0,C 180,E1 -4727.627,E2 -4727.627} C_VEL
LIN {X 0,Y 651.433,Z 347.434,A -85,B 0,C 180,E1 -4728.441,E2 -4728.441} C_VEL
LIN {X 0,Y 659.934,Z 369.917,A -85,B 0,C 180,E1 -4730.928,E2 -4730.928} C_VEL
LIN {X 0,Y 661.535,Z 374.738,A -85,B 0,C 180,E1 -4731.424,E2 -4731.424} C_VEL
LIN {X 0,Y 661.641,Z 376.516,A -85,B 0,C 180,E1 -4731.528,E2 -4731.528} C_VEL
LIN {X 0,Y 667.865,Z 402.872,A -85,B 0,C 180,E1 -4732.299,E2 -4732.299} C_VEL
LIN {X 0,Y 664.643,Z 668.434,A -85,B 0,C 180,E1 -4735.56,E2 -4735.56} C_VEL
LIN {X 0,Y 663.414,Z 767.858,A -85,B 0,C 180,E1 -4736.785,E2 -4736.785} C_VEL
LIN {X 0,Y 662.658,Z 793.274,A -85,B 0,C 180,E1 -4737.252,E2 -4737.252} C_VEL
LIN {X 0,Y 661.842,Z 814.057,A -85,B 0,C 180,E1 -4737.765,E2 -4737.765} C_VEL
LIN {X 0,Y 660.815,Z 837.255,A -85,B 0,C 180,E1 -4738.481,E2 -4738.481} C_VEL
LIN {X 0,Y 659.604,Z 859.334,A -85,B 0,C 180,E1 -4739.33,E2 -4739.33} C_VEL
LIN {X 0,Y 658.379,Z 881.272,A -85,B 0,C 180,E1 -4740.324,E2 -4740.324} C_VEL
LIN {X 0,Y 656.935,Z 903.117,A -85,B 0,C 180,E1 -4741.5,E2 -4741.5} C_VEL
LIN {X 0,Y 655.617,Z 923.649,A -85,B 0,C 180,E1 -4742.772,E2 -4742.772} C_VEL
LIN {X 0,Y 654.268,Z 943.217,A -85,B 0,C 180,E1 -4744.179,E2 -4744.179} C_VEL
LIN {X 0,Y 653.066,Z 961.203,A -85,B 0,C 180,E1 -4745.643,E2 -4745.643} C_VEL
LIN {X 0,Y 651.925,Z 978.603,A -85,B 0,C 180,E1 -4747.263,E2 -4747.263} C_VEL
LIN {X 0,Y 650.992,Z 993.629,A -85,B 0,C 180,E1 -4748.842,E2 -4748.842} C_VEL
LIN {X 0,Y 650.06,Z 1010.027,A -85,B 0,C 180,E1 -4750.809,E2 -4750.809} C_VEL
LIN {X 0,Y 649.428,Z 1022.519,A -85,B 0,C 180,E1 -4752.528,E2 -4752.528} C_VEL
LIN {X 0,Y 648.846,Z 1035.767,A -85,B 0,C 180,E1 -4754.63,E2 -4754.63} C_VEL
LIN {X 0,Y 648.494,Z 1045.563,A -85,B 0,C 180,E1 -4756.446,E2 -4756.446} C_VEL
LIN {X 0,Y 648.208,Z 1055.479,A -85,B 0,C 180,E1 -4758.612,E2 -4758.612} C_VEL
LIN {X 0,Y 648.055,Z 1062.514,A -85,B 0,C 180,E1 -4760.497,E2 -4760.497} C_VEL
LIN {X 0,Y 647.954,Z 1068.761,A -85,B 0,C 180,E1 -4762.552,E2 -4762.552} C_VEL
LIN {X 0,Y 647.924,Z 1073.496,A -85,B 0,C 180,E1 -4764.687,E2 -4764.687} C_VEL
LIN {X 0,Y 647.913,Z 1076.35,A -85,B 0,C 180,E1 -4766.549,E2 -4766.549} C_VEL
LIN {X 0,Y 647.905,Z 1078.192,A -85,B 0,C 180,E1 -4768.762,E2 -4768.762} C_VEL
LIN {X 0,Y 647.897,Z 1078.328,A -85,B 0,C 180,E1 -4770.707,E2 -4770.707} C_VEL
LIN {X 0,Y 647.907,Z 1077.157,A -85,B 0,C 180,E1 -4772.742,E2 -4772.742} C_VEL
LIN {X 0,Y 647.925,Z 1074.133,A -85,B 0,C 180,E1 -4774.958,E2 -4774.958} C_VEL
LIN {X 0,Y 647.94,Z 1070.276,A -85,B 0,C 180,E1 -4776.824,E2 -4776.824} C_VEL
LIN {X 0,Y 648.021,Z 1064.006,A -85,B 0,C 180,E1 -4779.062,E2 -4779.062} C_VEL
LIN {X 0,Y 648.158,Z 1057.25,A -85,B 0,C 180,E1 -4780.938,E2 -4780.938} C_VEL
LIN {X 0,Y 648.402,Z 1048.623,A -85,B 0,C 180,E1 -4782.941,E2 -4782.941} C_VEL
LIN {X 0,Y 648.764,Z 1037.835,A -85,B 0,C 180,E1 -4785.006,E2 -4785.006} C_VEL
LIN {X 0,Y 649.259,Z 1026.235,A -85,B 0,C 180,E1 -4786.922,E2 -4786.922} C_VEL
LIN {X 0,Y 649.923,Z 1012.35,A -85,B 0,C 180,E1 -4788.886,E2 -4788.886} C_VEL
LIN {X 0,Y 650.773,Z 997.755,A -85,B 0,C 180,E1 -4790.695,E2 -4790.695} C_VEL
LIN {X 0,Y 651.742,Z 981.381,A -85,B 0,C 180,E1 -4792.458,E2 -4792.458} C_VEL
LIN {X 0,Y 652.839,Z 964.771,A -85,B 0,C 180,E1 -4794.042,E2 -4794.042} C_VEL
LIN {X 0,Y 654.088,Z 945.648,A -85,B 0,C 180,E1 -4795.634,E2 -4795.634} C_VEL
LIN {X 0,Y 655.324,Z 927.727,A -85,B 0,C 180,E1 -4796.947,E2 -4796.947} C_VEL
LIN {X 0,Y 656.777,Z 905.546,A -85,B 0,C 180,E1 -4798.359,E2 -4798.359} C_VEL
LIN {X 0,Y 658.052,Z 885.844,A -85,B 0,C 180,E1 -4799.442,E2 -4799.442} C_VEL
LIN {X 0,Y 659.456,Z 862.306,A -85,B 0,C 180,E1 -4800.545,E2 -4800.545} C_VEL
LIN {X 0,Y 660.538,Z 842.394,A -85,B 0,C 180,E1 -4801.33,E2 -4801.33} C_VEL
LIN {X 0,Y 661.641,Z 818.851,A -85,B 0,C 180,E1 -4802.105,E2 -4802.105} C_VEL
LIN {X 0,Y 662.54,Z 796.094,A -85,B 0,C 180,E1 -4802.685,E2 -4802.685} C_VEL
LIN {X 0,Y 663.333,Z 772.593,A -85,B 0,C 180,E1 -4803.144,E2 -4803.144} C_VEL
LIN {X 0,Y 663.909,Z 733.531,A -85,B 0,C 180,E1 -4803.652,E2 -4803.652} C_VEL
LIN {X 0,Y 666.864,Z 481.94,A -85,B 0,C 180,E1 -4806.722,E2 -4806.722} C_VEL
LIN {X 0,Y 667.697,Z 401.371,A -85,B 0,C 180,E1 -4807.732,E2 -4807.732} C_VEL
LIN {X 0,Y 661.514,Z 375.529,A -85,B 0,C 180,E1 -4808.517,E2 -4808.517} C_VEL
LIN {X 0,Y 661.214,Z 373.349,A -85,B 0,C 180,E1 -4808.712,E2 -4808.712} C_VEL
LIN {X 0,Y 653.386,Z 352.647,A -85,B 0,C 180,E1 -4810.949,E2 -4810.949} C_VEL
LIN {X 0,Y 648.724,Z 340.426,A -85,B 0,C 180,E1 -4812.342,E2 -4812.342} C_VEL
LIN {X 0,Y 648.719,Z 340.427,A -85,B 0,C 180,E1 -4815.531,E2 -4815.531} C_VEL
LIN {X 0,Y 648.708,Z 340.423,A -85,B 0,C 180,E1 -4818.251,E2 -4818.251} C_VEL
LIN {X 0,Y 648.761,Z 340.422,A -85,B 0,C 180,E1 -4821.263,E2 -4821.263} C_VEL
LIN {X 0,Y 648.702,Z 340.422,A -85,B 0,C 180,E1 -4824.17,E2 -4824.17} C_VEL
LIN {X 0,Y 648.772,Z 340.416,A -85,B 0,C 180,E1 -4827.146,E2 -4827.146} C_VEL
LIN {X 0,Y 648.703,Z 340.419,A -85,B 0,C 180,E1 -4830.141,E2 -4830.141} C_VEL
LIN {X 0,Y 648.756,Z 340.407,A -85,B 0,C 180,E1 -4832.979,E2 -4832.979} C_VEL
LIN {X 0,Y 648.706,Z 340.412,A -85,B 0,C 180,E1 -4836.068,E2 -4836.068} C_VEL
LIN {X 0,Y 648.727,Z 340.418,A -85,B 0,C 180,E1 -4838.827,E2 -4838.827} C_VEL
LIN {X 0,Y 648.715,Z 340.421,A -85,B 0,C 180,E1 -4842.045,E2 -4842.045} C_VEL
LIN {X 0,Y 648.717,Z 340.415,A -85,B 0,C 180,E1 -4844.81,E2 -4844.81} C_VEL
LIN {X 0,Y 648.729,Z 340.422,A -85,B 0,C 180,E1 -4847.99,E2 -4847.99} C_VEL
LIN {X 0,Y 648.707,Z 340.407,A -85,B 0,C 180,E1 -4850.776,E2 -4850.776} C_VEL
LIN {X 0,Y 648.763,Z 340.418,A -85,B 0,C 180,E1 -4853.807,E2 -4853.807} C_VEL
LIN {X 0,Y 648.703,Z 340.416,A -85,B 0,C 180,E1 -4856.731,E2 -4856.731} C_VEL
LIN {X 0,Y 648.775,Z 340.412,A -85,B 0,C 180,E1 -4859.735,E2 -4859.735} C_VEL
LIN {X 0,Y 648.704,Z 340.42,A -85,B 0,C 180,E1 -4862.739,E2 -4862.739} C_VEL
LIN {X 0,Y 648.768,Z 340.409,A -85,B 0,C 180,E1 -4865.661,E2 -4865.661} C_VEL
LIN {X 0,Y 648.706,Z 340.421,A -85,B 0,C 180,E1 -4868.688,E2 -4868.688} C_VEL
LIN {X 0,Y 648.747,Z 340.403,A -85,B 0,C 180,E1 -4871.558,E2 -4871.558} C_VEL
LIN {X 0,Y 648.713,Z 340.417,A -85,B 0,C 180,E1 -4874.642,E2 -4874.642} C_VEL
LIN {X 0,Y 648.725,Z 340.413,A -85,B 0,C 180,E1 -4877.432,E2 -4877.432} C_VEL
LIN {X 0,Y 648.718,Z 340.411,A -85,B 0,C 180,E1 -4880.677,E2 -4880.677} C_VEL
LIN {X 0,Y 648.717,Z 340.419,A -85,B 0,C 180,E1 -4883.432,E2 -4883.432} C_VEL
LIN {X 0,Y 648.732,Z 340.423,A -85,B 0,C 180,E1 -4886.649,E2 -4886.649} C_VEL
LIN {X 0,Y 648.712,Z 340.409,A -85,B 0,C 180,E1 -4889.452,E2 -4889.452} C_VEL
LIN {X 0,Y 648.756,Z 340.414,A -85,B 0,C 180,E1 -4892.541,E2 -4892.541} C_VEL
LIN {X 0,Y 648.71,Z 340.42,A -85,B 0,C 180,E1 -4895.419,E2 -4895.419} C_VEL
LIN {X 0,Y 648.773,Z 340.422,A -85,B 0,C 180,E1 -4898.51,E2 -4898.51} C_VEL
LIN {X 0,Y 648.707,Z 340.424,A -85,B 0,C 180,E1 -4901.395,E2 -4901.395} C_VEL
LIN {X 0,Y 648.773,Z 340.412,A -85,B 0,C 180,E1 -4902.429,E2 -4902.429} C_VEL
LIN {X 0,Y 647.756,Z 340.524,A -85,B 0,C 180,E1 -4903.109,E2 -4903.109} C_VEL
LIN {X 0,Y 641.295,Z 341.322,A -85,B 0,C 180,E1 -4905.016,E2 -4905.016} C_VEL
LIN {X 0,Y 640.768,Z 341.399,A -85,B 0,C 180,E1 -4905.513,E2 -4905.513} C_VEL
LIN {X 0,Y 640.837,Z 341.402,A -85,B 0,C 180,E1 -4908.499,E2 -4908.499} C_VEL
LIN {X 0,Y 640.79,Z 341.545,A -85,B 0,C 180,E1 -4911.365,E2 -4911.365} C_VEL
LIN {X 0,Y 643.877,Z 349.627,A -85,B 0,C 180,E1 -4912.318,E2 -4912.318} C_VEL
LIN {X 0,Y 658.867,Z 374.361,A -85,B 0,C 180,E1 -4913.729,E2 -4913.729} C_VEL
LIN {X 0,Y 661.548,Z 379.54,A -85,B 0,C 180,E1 -4913.983,E2 -4913.983} C_VEL
LIN {X 0,Y 658.385,Z 617.08,A -85,B 0,C 180,E1 -4916.94,E2 -4916.94} C_VEL
LIN {X 0,Y 656.757,Z 738.068,A -85,B 0,C 180,E1 -4918.443,E2 -4918.443} C_VEL
LIN {X 0,Y 655.957,Z 763.521,A -85,B 0,C 180,E1 -4918.915,E2 -4918.915} C_VEL
LIN {X 0,Y 655.09,Z 784.002,A -85,B 0,C 180,E1 -4919.425,E2 -4919.425} C_VEL
LIN {X 0,Y 654.039,Z 806.034,A -85,B 0,C 180,E1 -4920.107,E2 -4920.107} C_VEL
LIN {X 0,Y 652.714,Z 827.923,A -85,B 0,C 180,E1 -4920.948,E2 -4920.948} C_VEL
LIN {X 0,Y 651.447,Z 848.647,A -85,B 0,C 180,E1 -4921.887,E2 -4921.887} C_VEL
LIN {X 0,Y 649.878,Z 871.49,A -85,B 0,C 180,E1 -4923.106,E2 -4923.106} C_VEL
LIN {X 0,Y 648.51,Z 890.461,A -85,B 0,C 180,E1 -4924.277,E2 -4924.277} C_VEL
LIN {X 0,Y 647.011,Z 911.25,A -85,B 0,C 180,E1 -4925.754,E2 -4925.754} C_VEL
LIN {X 0,Y 645.766,Z 928.204,A -85,B 0,C 180,E1 -4927.13,E2 -4927.13} C_VEL
LIN {X 0,Y 644.461,Z 946.619,A -85,B 0,C 180,E1 -4928.823,E2 -4928.823} C_VEL
LIN {X 0,Y 643.38,Z 962.356,A -85,B 0,C 180,E1 -4930.48,E2 -4930.48} C_VEL
LIN {X 0,Y 642.423,Z 977.898,A -85,B 0,C 180,E1 -4932.332,E2 -4932.332} C_VEL
LIN {X 0,Y 641.632,Z 991.301,A -85,B 0,C 180,E1 -4934.174,E2 -4934.174} C_VEL
LIN {X 0,Y 641.024,Z 1004.152,A -85,B 0,C 180,E1 -4936.193,E2 -4936.193} C_VEL
LIN {X 0,Y 640.573,Z 1014.97,A -85,B 0,C 180,E1 -4938.201,E2 -4938.201} C_VEL
LIN {X 0,Y 640.272,Z 1024.604,A -85,B 0,C 180,E1 -4940.29,E2 -4940.29} C_VEL
LIN {X 0,Y 640.067,Z 1032.335,A -85,B 0,C 180,E1 -4942.37,E2 -4942.37} C_VEL
LIN {X 0,Y 639.965,Z 1038.079,A -85,B 0,C 180,E1 -4944.261,E2 -4944.261} C_VEL
LIN {X 0,Y 639.916,Z 1043.212,A -85,B 0,C 180,E1 -4946.506,E2 -4946.506} C_VEL
LIN {X 0,Y 639.913,Z 1046.145,A -85,B 0,C 180,E1 -4948.388,E2 -4948.388} C_VEL
LIN {X 0,Y 639.9,Z 1048.112,A -85,B 0,C 180,E1 -4950.537,E2 -4950.537} C_VEL
LIN {X 0,Y 639.895,Z 1048.347,A -85,B 0,C 180,E1 -4952.687,E2 -4952.687} C_VEL
LIN {X 0,Y 639.898,Z 1047.279,A -85,B 0,C 180,E1 -4954.661,E2 -4954.661} C_VEL
LIN {X 0,Y 639.917,Z 1044.407,A -85,B 0,C 180,E1 -4956.91,E2 -4956.91} C_VEL
LIN {X 0,Y 639.946,Z 1040.613,A -85,B 0,C 180,E1 -4958.808,E2 -4958.808} C_VEL
LIN {X 0,Y 640.019,Z 1034.786,A -85,B 0,C 180,E1 -4960.988,E2 -4960.988} C_VEL
LIN {X 0,Y 640.168,Z 1027.729,A -85,B 0,C 180,E1 -4962.998,E2 -4962.998} C_VEL
LIN {X 0,Y 640.412,Z 1019.823,A -85,B 0,C 180,E1 -4964.88,E2 -4964.88} C_VEL
LIN {X 0,Y 640.82,Z 1008.851,A -85,B 0,C 180,E1 -4967.058,E2 -4967.058} C_VEL
LIN {X 0,Y 641.314,Z 997.845,A -85,B 0,C 180,E1 -4968.923,E2 -4968.923} C_VEL
LIN {X 0,Y 642.053,Z 983.699,A -85,B 0,C 180,E1 -4970.989,E2 -4970.989} C_VEL
LIN {X 0,Y 642.904,Z 969.922,A -85,B 0,C 180,E1 -4972.738,E2 -4972.738} C_VEL
LIN {X 0,Y 644.05,Z 952.357,A -85,B 0,C 180,E1 -4974.685,E2 -4974.685} C_VEL
LIN {X 0,Y 645.16,Z 936.633,A -85,B 0,C 180,E1 -4976.213,E2 -4976.213} C_VEL
LIN {X 0,Y 646.621,Z 916.353,A -85,B 0,C 180,E1 -4977.939,E2 -4977.939} C_VEL
LIN {X 0,Y 647.915,Z 898.903,A -85,B 0,C 180,E1 -4979.238,E2 -4979.238} C_VEL
LIN {X 0,Y 649.455,Z 877.42,A -85,B 0,C 180,E1 -4980.637,E2 -4980.637} C_VEL
LIN {X 0,Y 650.753,Z 858.498,A -85,B 0,C 180,E1 -4981.701,E2 -4981.701} C_VEL
LIN {X 0,Y 652.23,Z 836.818,A -85,B 0,C 180,E1 -4982.763,E2 -4982.763} C_VEL
LIN {X 0,Y 653.53,Z 814.727,A -85,B 0,C 180,E1 -4983.663,E2 -4983.663} C_VEL
LIN {X 0,Y 654.64,Z 793.649,A -85,B 0,C 180,E1 -4984.385,E2 -4984.385} C_VEL
LIN {X 0,Y 655.721,Z 768.897,A -85,B 0,C 180,E1 -4985.054,E2 -4985.054} C_VEL
LIN {X 0,Y 656.498,Z 747.393,A -85,B 0,C 180,E1 -4985.494,E2 -4985.494} C_VEL
LIN {X 0,Y 657.137,Z 716.349,A -85,B 0,C 180,E1 -4985.934,E2 -4985.934} C_VEL
LIN {X 0,Y 660.441,Z 462.018,A -85,B 0,C 180,E1 -4989.071,E2 -4989.071} C_VEL
LIN {X 0,Y 661.384,Z 378.795,A -85,B 0,C 180,E1 -4990.128,E2 -4990.128} C_VEL
LIN {X 0,Y 649.906,Z 359.323,A -85,B 0,C 180,E1 -4991.207,E2 -4991.207} C_VEL
LIN {X 0,Y 643.631,Z 348.945,A -85,B 0,C 180,E1 -4991.848,E2 -4991.848} C_VEL
LIN {X 0,Y 640.777,Z 341.41,A -85,B 0,C 180,E1 -4992.81,E2 -4992.81} C_VEL
LIN {X 0,Y 640.799,Z 341.403,A -85,B 0,C 180,E1 -4996,E2 -4996} C_VEL
LIN {X 0,Y 640.766,Z 341.392,A -85,B 0,C 180,E1 -4998.813,E2 -4998.813} C_VEL
LIN {X 0,Y 640.826,Z 341.406,A -85,B 0,C 180,E1 -5001.85,E2 -5001.85} C_VEL
LIN {X 0,Y 640.765,Z 341.385,A -85,B 0,C 180,E1 -5004.843,E2 -5004.843} C_VEL
LIN {X 0,Y 640.829,Z 341.399,A -85,B 0,C 180,E1 -5007.913,E2 -5007.913} C_VEL
LIN {X 0,Y 640.766,Z 341.409,A -85,B 0,C 180,E1 -5010.865,E2 -5010.865} C_VEL
LIN {X 0,Y 640.833,Z 341.403,A -85,B 0,C 180,E1 -5013.796,E2 -5013.796} C_VEL
LIN {X 0,Y 640.766,Z 341.41,A -85,B 0,C 180,E1 -5016.844,E2 -5016.844} C_VEL
LIN {X 0,Y 640.822,Z 341.407,A -85,B 0,C 180,E1 -5019.733,E2 -5019.733} C_VEL
LIN {X 0,Y 640.767,Z 341.404,A -85,B 0,C 180,E1 -5022.847,E2 -5022.847} C_VEL
LIN {X 0,Y 640.808,Z 341.403,A -85,B 0,C 180,E1 -5025.727,E2 -5025.727} C_VEL
LIN {X 0,Y 640.773,Z 341.406,A -85,B 0,C 180,E1 -5028.843,E2 -5028.843} C_VEL
LIN {X 0,Y 640.787,Z 341.408,A -85,B 0,C 180,E1 -5031.656,E2 -5031.656} C_VEL
LIN {X 0,Y 640.781,Z 341.402,A -85,B 0,C 180,E1 -5034.807,E2 -5034.807} C_VEL
LIN {X 0,Y 640.774,Z 341.41,A -85,B 0,C 180,E1 -5037.585,E2 -5037.585} C_VEL
LIN {X 0,Y 640.791,Z 341.407,A -85,B 0,C 180,E1 -5040.805,E2 -5040.805} C_VEL
LIN {X 0,Y 640.767,Z 341.402,A -85,B 0,C 180,E1 -5043.579,E2 -5043.579} C_VEL
LIN {X 0,Y 640.825,Z 341.394,A -85,B 0,C 180,E1 -5046.63,E2 -5046.63} C_VEL
LIN {X 0,Y 640.764,Z 341.41,A -85,B 0,C 180,E1 -5049.525,E2 -5049.525} C_VEL
LIN {X 0,Y 640.834,Z 341.405,A -85,B 0,C 180,E1 -5052.526,E2 -5052.526} C_VEL
LIN {X 0,Y 640.764,Z 341.398,A -85,B 0,C 180,E1 -5055.476,E2 -5055.476} C_VEL
LIN {X 0,Y 640.816,Z 341.405,A -85,B 0,C 180,E1 -5058.372,E2 -5058.372} C_VEL
LIN {X 0,Y 640.772,Z 341.408,A -85,B 0,C 180,E1 -5061.417,E2 -5061.417} C_VEL
LIN {X 0,Y 640.789,Z 341.403,A -85,B 0,C 180,E1 -5064.229,E2 -5064.229} C_VEL
LIN {X 0,Y 640.777,Z 341.403,A -85,B 0,C 180,E1 -5067.408,E2 -5067.408} C_VEL
LIN {X 0,Y 640.771,Z 341.409,A -85,B 0,C 180,E1 -5070.06,E2 -5070.06} C_VEL
LIN {X 0,Y 640.807,Z 341.409,A -85,B 0,C 180,E1 -5073.209,E2 -5073.209} C_VEL
LIN {X 0,Y 640.766,Z 341.412,A -85,B 0,C 180,E1 -5076.068,E2 -5076.068} C_VEL
LIN {X 0,Y 640.826,Z 341.407,A -85,B 0,C 180,E1 -5079.152,E2 -5079.152} C_VEL
LIN {X 0,Y 640.763,Z 341.411,A -85,B 0,C 180,E1 -5082.031,E2 -5082.031} C_VEL
LIN {X 0,Y 640.833,Z 341.407,A -85,B 0,C 180,E1 -5085.024,E2 -5085.024} C_VEL
LIN {X 0,Y 640.837,Z 341.434,A -85,B 0,C 180,E1 -5087.077,E2 -5087.077} C_VEL
LIN {X 0,Y 648.847,Z 362.263,A -85,B 0,C 180,E1 -5089.508,E2 -5089.508} C_VEL
LIN {X 0,Y 654.011,Z 376.024,A -85,B 0,C 180,E1 -5090.991,E2 -5090.991} C_VEL
LIN {X 0,Y 655.595,Z 379.441,A -85,B 0,C 180,E1 -5091.15,E2 -5091.15} C_VEL
LIN {X 0,Y 661.495,Z 404.617,A -85,B 0,C 180,E1 -5091.898,E2 -5091.898} C_VEL
LIN {X 0,Y 657.99,Z 671.647,A -85,B 0,C 180,E1 -5095.207,E2 -5095.207} C_VEL
LIN {X 0,Y 656.699,Z 767.707,A -85,B 0,C 180,E1 -5096.401,E2 -5096.401} C_VEL
LIN {X 0,Y 655.892,Z 793.05,A -85,B 0,C 180,E1 -5096.871,E2 -5096.871} C_VEL
LIN {X 0,Y 655.03,Z 813.506,A -85,B 0,C 180,E1 -5097.379,E2 -5097.379} C_VEL
LIN {X 0,Y 653.952,Z 836.425,A -85,B 0,C 180,E1 -5098.086,E2 -5098.086} C_VEL
LIN {X 0,Y 652.608,Z 859.258,A -85,B 0,C 180,E1 -5098.965,E2 -5098.965} C_VEL
LIN {X 0,Y 651.357,Z 880.271,A -85,B 0,C 180,E1 -5099.92,E2 -5099.92} C_VEL
LIN {X 0,Y 649.815,Z 902.324,A -85,B 0,C 180,E1 -5101.109,E2 -5101.109} C_VEL
LIN {X 0,Y 648.444,Z 921.455,A -85,B 0,C 180,E1 -5102.296,E2 -5102.296} C_VEL
LIN {X 0,Y 646.957,Z 941.998,A -85,B 0,C 180,E1 -5103.767,E2 -5103.767} C_VEL
LIN {X 0,Y 645.698,Z 959.036,A -85,B 0,C 180,E1 -5105.155,E2 -5105.155} C_VEL
LIN {X 0,Y 644.315,Z 978.602,A -85,B 0,C 180,E1 -5106.979,E2 -5106.979} C_VEL
LIN {X 0,Y 643.282,Z 993.856,A -85,B 0,C 180,E1 -5108.601,E2 -5108.601} C_VEL
LIN {X 0,Y 642.297,Z 1009.819,A -85,B 0,C 180,E1 -5110.54,E2 -5110.54} C_VEL
LIN {X 0,Y 641.577,Z 1022.517,A -85,B 0,C 180,E1 -5112.308,E2 -5112.308} C_VEL
LIN {X 0,Y 640.946,Z 1035.769,A -85,B 0,C 180,E1 -5114.435,E2 -5114.435} C_VEL
LIN {X 0,Y 640.557,Z 1045.561,A -85,B 0,C 180,E1 -5116.275,E2 -5116.275} C_VEL
LIN {X 0,Y 640.244,Z 1055.479,A -85,B 0,C 180,E1 -5118.469,E2 -5118.469} C_VEL
LIN {X 0,Y 640.064,Z 1062.514,A -85,B 0,C 180,E1 -5120.378,E2 -5120.378} C_VEL
LIN {X 0,Y 639.958,Z 1068.507,A -85,B 0,C 180,E1 -5122.368,E2 -5122.368} C_VEL
LIN {X 0,Y 639.926,Z 1073.336,A -85,B 0,C 180,E1 -5124.531,E2 -5124.531} C_VEL
LIN {X 0,Y 639.908,Z 1076.238,A -85,B 0,C 180,E1 -5126.417,E2 -5126.417} C_VEL
LIN {X 0,Y 639.894,Z 1078.146,A -85,B 0,C 180,E1 -5128.567,E2 -5128.567} C_VEL
LIN {X 0,Y 639.894,Z 1078.35,A -85,B 0,C 180,E1 -5130.627,E2 -5130.627} C_VEL
LIN {X 0,Y 639.907,Z 1077.293,A -85,B 0,C 180,E1 -5132.597,E2 -5132.597} C_VEL
LIN {X 0,Y 639.924,Z 1074.451,A -85,B 0,C 180,E1 -5134.84,E2 -5134.84} C_VEL
LIN {X 0,Y 639.935,Z 1070.689,A -85,B 0,C 180,E1 -5136.73,E2 -5136.73} C_VEL
LIN {X 0,Y 640.008,Z 1065.202,A -85,B 0,C 180,E1 -5138.807,E2 -5138.807} C_VEL
LIN {X 0,Y 640.169,Z 1057.956,A -85,B 0,C 180,E1 -5140.894,E2 -5140.894} C_VEL
LIN {X 0,Y 640.404,Z 1049.938,A -85,B 0,C 180,E1 -5142.81,E2 -5142.81} C_VEL
LIN {X 0,Y 640.813,Z 1038.847,A -85,B 0,C 180,E1 -5145.015,E2 -5145.015} C_VEL
LIN {X 0,Y 641.3,Z 1027.973,A -85,B 0,C 180,E1 -5146.858,E2 -5146.858} C_VEL
LIN {X 0,Y 642.038,Z 1014.022,A -85,B 0,C 180,E1 -5148.901,E2 -5148.901} C_VEL
LIN {X 0,Y 642.841,Z 1000.849,A -85,B 0,C 180,E1 -5150.581,E2 -5150.581} C_VEL
LIN {X 0,Y 643.933,Z 984.157,A -85,B 0,C 180,E1 -5152.457,E2 -5152.457} C_VEL
LIN {X 0,Y 645.033,Z 968.318,A -85,B 0,C 180,E1 -5154.011,E2 -5154.011} C_VEL
LIN {X 0,Y 646.361,Z 950.193,A -85,B 0,C 180,E1 -5155.594,E2 -5155.594} C_VEL
LIN {X 0,Y 647.746,Z 931.053,A -85,B 0,C 180,E1 -5157.04,E2 -5157.04} C_VEL
LIN {X 0,Y 649.228,Z 911.161,A -85,B 0,C 180,E1 -5158.368,E2 -5158.368} C_VEL
LIN {X 0,Y 650.632,Z 890.298,A -85,B 0,C 180,E1 -5159.561,E2 -5159.561} C_VEL
LIN {X 0,Y 651.972,Z 870.217,A -85,B 0,C 180,E1 -5160.557,E2 -5160.557} C_VEL
LIN {X 0,Y 653.351,Z 847.074,A -85,B 0,C 180,E1 -5161.522,E2 -5161.522} C_VEL
LIN {X 0,Y 654.406,Z 826.841,A -85,B 0,C 180,E1 -5162.225,E2 -5162.225} C_VEL
LIN {X 0,Y 655.479,Z 803.653,A -85,B 0,C 180,E1 -5162.889,E2 -5162.889} C_VEL
LIN {X 0,Y 656.33,Z 779.724,A -85,B 0,C 180,E1 -5163.397,E2 -5163.397} C_VEL
LIN {X 0,Y 656.97,Z 755.117,A -85,B 0,C 180,E1 -5163.775,E2 -5163.775} C_VEL
LIN {X 0,Y 660.095,Z 506.842,A -85,B 0,C 180,E1 -5166.827,E2 -5166.827} C_VEL
LIN {X 0,Y 661.336,Z 403.158,A -85,B 0,C 180,E1 -5168.133,E2 -5168.133} C_VEL
LIN {X 0,Y 655.032,Z 377.89,A -85,B 0,C 180,E1 -5168.911,E2 -5168.911} C_VEL
LIN {X 0,Y 653.661,Z 375.262,A -85,B 0,C 180,E1 -5169.067,E2 -5169.067} C_VEL
LIN {X 0,Y 645.884,Z 354.531,A -85,B 0,C 180,E1 -5171.338,E2 -5171.338} C_VEL
LIN {X 0,Y 640.832,Z 341.411,A -85,B 0,C 180,E1 -5172.866,E2 -5172.866} C_VEL
LIN {X 0,Y 640.763,Z 341.414,A -85,B 0,C 180,E1 -5175.895,E2 -5175.895} C_VEL
LIN {X 0,Y 640.837,Z 341.408,A -85,B 0,C 180,E1 -5178.905,E2 -5178.905} C_VEL
LIN {X 0,Y 640.764,Z 341.409,A -85,B 0,C 180,E1 -5181.947,E2 -5181.947} C_VEL
LIN {X 0,Y 640.817,Z 341.408,A -85,B 0,C 180,E1 -5184.847,E2 -5184.847} C_VEL
LIN {X 0,Y 640.766,Z 341.408,A -85,B 0,C 180,E1 -5187.957,E2 -5187.957} C_VEL
LIN {X 0,Y 640.795,Z 341.406,A -85,B 0,C 180,E1 -5190.764,E2 -5190.764} C_VEL
LIN {X 0,Y 640.777,Z 341.41,A -85,B 0,C 180,E1 -5193.893,E2 -5193.893} C_VEL
LIN {X 0,Y 640.777,Z 341.397,A -85,B 0,C 180,E1 -5196.65,E2 -5196.65} C_VEL
LIN {X 0,Y 640.782,Z 341.403,A -85,B 0,C 180,E1 -5199.922,E2 -5199.922} C_VEL
LIN {X 0,Y 640.777,Z 341.406,A -85,B 0,C 180,E1 -5202.753,E2 -5202.753} C_VEL
LIN {X 0,Y 640.784,Z 341.403,A -85,B 0,C 180,E1 -5206.003,E2 -5206.003} C_VEL
LIN {X 0,Y 640.77,Z 341.407,A -85,B 0,C 180,E1 -5208.752,E2 -5208.752} C_VEL
LIN {X 0,Y 640.804,Z 341.408,A -85,B 0,C 180,E1 -5211.927,E2 -5211.927} C_VEL
LIN {X 0,Y 640.766,Z 341.401,A -85,B 0,C 180,E1 -5214.717,E2 -5214.717} C_VEL
LIN {X 0,Y 640.831,Z 341.407,A -85,B 0,C 180,E1 -5217.764,E2 -5217.764} C_VEL
LIN {X 0,Y 640.763,Z 341.394,A -85,B 0,C 180,E1 -5220.715,E2 -5220.715} C_VEL
LIN {X 0,Y 640.831,Z 341.406,A -85,B 0,C 180,E1 -5223.668,E2 -5223.668} C_VEL
LIN {X 0,Y 640.765,Z 341.403,A -85,B 0,C 180,E1 -5226.721,E2 -5226.721} C_VEL
LIN {X 0,Y 640.819,Z 341.405,A -85,B 0,C 180,E1 -5229.611,E2 -5229.611} C_VEL
LIN {X 0,Y 640.771,Z 341.409,A -85,B 0,C 180,E1 -5232.71,E2 -5232.71} C_VEL
LIN {X 0,Y 640.792,Z 341.402,A -85,B 0,C 180,E1 -5235.476,E2 -5235.476} C_VEL
LIN {X 0,Y 640.78,Z 341.41,A -85,B 0,C 180,E1 -5238.656,E2 -5238.656} C_VEL
LIN {X 0,Y 640.779,Z 341.397,A -85,B 0,C 180,E1 -5241.416,E2 -5241.416} C_VEL
LIN {X 0,Y 640.79,Z 341.4,A -85,B 0,C 180,E1 -5244.622,E2 -5244.622} C_VEL
LIN {X 0,Y 640.775,Z 341.408,A -85,B 0,C 180,E1 -5247.409,E2 -5247.409} C_VEL
LIN {X 0,Y 640.814,Z 341.405,A -85,B 0,C 180,E1 -5250.536,E2 -5250.536} C_VEL
LIN {X 0,Y 640.769,Z 341.4,A -85,B 0,C 180,E1 -5253.425,E2 -5253.425} C_VEL
LIN {X 0,Y 640.823,Z 341.401,A -85,B 0,C 180,E1 -5256.528,E2 -5256.528} C_VEL
LIN {X 0,Y 640.767,Z 341.406,A -85,B 0,C 180,E1 -5259.428,E2 -5259.428} C_VEL
LIN {X 0,Y 640.834,Z 341.399,A -85,B 0,C 180,E1 -5262.437,E2 -5262.437} C_VEL
LIN {X 0,Y 640.768,Z 341.396,A -85,B 0,C 180,E1 -5265.396,E2 -5265.396} C_VEL
LIN {X 0,Y 640.768,Z 341.399,A -85,B 0,C 180,E1 -5265.513,E2 -5265.513} C_VEL
LIN {X 0,Y 639.803,Z 341.532,A -85,B 0,C 180,E1 -5266.201,E2 -5266.201} C_VEL
LIN {X 0,Y 633.446,Z 342.32,A -85,B 0,C 180,E1 -5268.133,E2 -5268.133} C_VEL
LIN {X 0,Y 632.899,Z 342.393,A -85,B 0,C 180,E1 -5268.635,E2 -5268.635} C_VEL
LIN {X 0,Y 632.911,Z 342.613,A -85,B 0,C 180,E1 -5270.839,E2 -5270.839} C_VEL
LIN {X 0,Y 635.679,Z 349.892,A -85,B 0,C 180,E1 -5271.712,E2 -5271.712} C_VEL
LIN {X 0,Y 653.275,Z 378.692,A -85,B 0,C 180,E1 -5273.398,E2 -5273.398} C_VEL
LIN {X 0,Y 655.217,Z 382.638,A -85,B 0,C 180,E1 -5273.588,E2 -5273.588} C_VEL
LIN {X 0,Y 651.805,Z 620.683,A -85,B 0,C 180,E1 -5276.577,E2 -5276.577} C_VEL
LIN {X 0,Y 650.1,Z 738.3,A -85,B 0,C 180,E1 -5278.053,E2 -5278.053} C_VEL
LIN {X 0,Y 649.255,Z 763.745,A -85,B 0,C 180,E1 -5278.528,E2 -5278.528} C_VEL
LIN {X 0,Y 648.345,Z 784.012,A -85,B 0,C 180,E1 -5279.037,E2 -5279.037} C_VEL
LIN {X 0,Y 647.226,Z 806.04,A -85,B 0,C 180,E1 -5279.723,E2 -5279.723} C_VEL
LIN {X 0,Y 645.756,Z 828.772,A -85,B 0,C 180,E1 -5280.604,E2 -5280.604} C_VEL
LIN {X 0,Y 644.399,Z 849.399,A -85,B 0,C 180,E1 -5281.552,E2 -5281.552} C_VEL
LIN {X 0,Y 642.764,Z 871.198,A -85,B 0,C 180,E1 -5282.734,E2 -5282.734} C_VEL
LIN {X 0,Y 641.223,Z 890.882,A -85,B 0,C 180,E1 -5283.963,E2 -5283.963} C_VEL
LIN {X 0,Y 639.565,Z 912.066,A -85,B 0,C 180,E1 -5285.491,E2 -5285.491} C_VEL
LIN {X 0,Y 638.248,Z 928.795,A -85,B 0,C 180,E1 -5286.869,E2 -5286.869} C_VEL
LIN {X 0,Y 636.792,Z 947.66,A -85,B 0,C 180,E1 -5288.636,E2 -5288.636} C_VEL
LIN {X 0,Y 635.693,Z 962.6,A -85,B 0,C 180,E1 -5290.234,E2 -5290.234} C_VEL
LIN {X 0,Y 634.597,Z 978.807,A -85,B 0,C 180,E1 -5292.201,E2 -5292.201} C_VEL
LIN {X 0,Y 633.792,Z 991.484,A -85,B 0,C 180,E1 -5293.973,E2 -5293.973} C_VEL
LIN {X 0,Y 633.129,Z 1004.305,A -85,B 0,C 180,E1 -5296.017,E2 -5296.017} C_VEL
LIN {X 0,Y 632.653,Z 1014.647,A -85,B 0,C 180,E1 -5297.958,E2 -5297.958} C_VEL
LIN {X 0,Y 632.324,Z 1023.928,A -85,B 0,C 180,E1 -5299.983,E2 -5299.983} C_VEL
LIN {X 0,Y 632.091,Z 1031.819,A -85,B 0,C 180,E1 -5302.09,E2 -5302.09} C_VEL
LIN {X 0,Y 631.988,Z 1037.646,A -85,B 0,C 180,E1 -5304.006,E2 -5304.006} C_VEL
LIN {X 0,Y 631.929,Z 1042.939,A -85,B 0,C 180,E1 -5306.28,E2 -5306.28} C_VEL
LIN {X 0,Y 631.914,Z 1046.063,A -85,B 0,C 180,E1 -5308.277,E2 -5308.277} C_VEL
LIN {X 0,Y 631.902,Z 1047.932,A -85,B 0,C 180,E1 -5310.272,E2 -5310.272} C_VEL
LIN {X 0,Y 631.893,Z 1048.385,A -85,B 0,C 180,E1 -5312.539,E2 -5312.539} C_VEL
LIN {X 0,Y 631.905,Z 1047.464,A -85,B 0,C 180,E1 -5314.447,E2 -5314.447} C_VEL
LIN {X 0,Y 631.923,Z 1044.999,A -85,B 0,C 180,E1 -5316.633,E2 -5316.633} C_VEL
LIN {X 0,Y 631.944,Z 1040.969,A -85,B 0,C 180,E1 -5318.737,E2 -5318.737} C_VEL
LIN {X 0,Y 632.006,Z 1036.026,A -85,B 0,C 180,E1 -5320.667,E2 -5320.667} C_VEL
LIN {X 0,Y 632.182,Z 1028.337,A -85,B 0,C 180,E1 -5322.979,E2 -5322.979} C_VEL
LIN {X 0,Y 632.43,Z 1020.718,A -85,B 0,C 180,E1 -5324.84,E2 -5324.84} C_VEL
LIN {X 0,Y 632.854,Z 1010.256,A -85,B 0,C 180,E1 -5326.995,E2 -5326.995} C_VEL
LIN {X 0,Y 633.396,Z 998.832,A -85,B 0,C 180,E1 -5328.977,E2 -5328.977} C_VEL
LIN {X 0,Y 634.177,Z 985.19,A -85,B 0,C 180,E1 -5331.03,E2 -5331.03} C_VEL
LIN {X 0,Y 635.064,Z 971.658,A -85,B 0,C 180,E1 -5332.788,E2 -5332.788} C_VEL
LIN {X 0,Y 636.229,Z 955.363,A -85,B 0,C 180,E1 -5334.662,E2 -5334.662} C_VEL
LIN {X 0,Y 637.495,Z 938.385,A -85,B 0,C 180,E1 -5336.351,E2 -5336.351} C_VEL
LIN {X 0,Y 638.921,Z 920.3,A -85,B 0,C 180,E1 -5337.95,E2 -5337.95} C_VEL
LIN {X 0,Y 640.414,Z 901.338,A -85,B 0,C 180,E1 -5339.399,E2 -5339.399} C_VEL
LIN {X 0,Y 641.967,Z 881.759,A -85,B 0,C 180,E1 -5340.722,E2 -5340.722} C_VEL
LIN {X 0,Y 643.591,Z 859.914,A -85,B 0,C 180,E1 -5341.991,E2 -5341.991} C_VEL
LIN {X 0,Y 645.086,Z 839.544,A -85,B 0,C 180,E1 -5343.012,E2 -5343.012} C_VEL
LIN {X 0,Y 646.555,Z 816.902,A -85,B 0,C 180,E1 -5343.964,E2 -5343.964} C_VEL
LIN {X 0,Y 647.698,Z 796.749,A -85,B 0,C 180,E1 -5344.672,E2 -5344.672} C_VEL
LIN {X 0,Y 648.85,Z 773.049,A -85,B 0,C 180,E1 -5345.349,E2 -5345.349} C_VEL
LIN {X 0,Y 649.724,Z 750.211,A -85,B 0,C 180,E1 -5345.836,E2 -5345.836} C_VEL
LIN {X 0,Y 650.389,Z 725.478,A -85,B 0,C 180,E1 -5346.218,E2 -5346.218} C_VEL
LIN {X 0,Y 653.922,Z 472.185,A -85,B 0,C 180,E1 -5349.368,E2 -5349.368} C_VEL
LIN {X 0,Y 655.065,Z 381.929,A -85,B 0,C 180,E1 -5350.522,E2 -5350.522} C_VEL
LIN {X 0,Y 644.365,Z 363.809,A -85,B 0,C 180,E1 -5351.554,E2 -5351.554} C_VEL
LIN {X 0,Y 635.544,Z 349.449,A -85,B 0,C 180,E1 -5352.449,E2 -5352.449} C_VEL
LIN {X 0,Y 632.89,Z 342.397,A -85,B 0,C 180,E1 -5353.375,E2 -5353.375} C_VEL
LIN {X 0,Y 632.83,Z 342.395,A -85,B 0,C 180,E1 -5356.457,E2 -5356.457} C_VEL
LIN {X 0,Y 632.893,Z 342.367,A -85,B 0,C 180,E1 -5359.457,E2 -5359.457} C_VEL
LIN {X 0,Y 632.83,Z 342.398,A -85,B 0,C 180,E1 -5362.532,E2 -5362.532} C_VEL
LIN {X 0,Y 632.876,Z 342.376,A -85,B 0,C 180,E1 -5365.445,E2 -5365.445} C_VEL
LIN {X 0,Y 632.831,Z 342.39,A -85,B 0,C 180,E1 -5368.573,E2 -5368.573} C_VEL
LIN {X 0,Y 632.86,Z 342.394,A -85,B 0,C 180,E1 -5371.398,E2 -5371.398} C_VEL
LIN {X 0,Y 632.837,Z 342.39,A -85,B 0,C 180,E1 -5374.547,E2 -5374.547} C_VEL
LIN {X 0,Y 632.843,Z 342.401,A -85,B 0,C 180,E1 -5377.327,E2 -5377.327} C_VEL
LIN {X 0,Y 632.841,Z 342.396,A -85,B 0,C 180,E1 -5380.622,E2 -5380.622} C_VEL
LIN {X 0,Y 632.847,Z 342.396,A -85,B 0,C 180,E1 -5383.477,E2 -5383.477} C_VEL
LIN {X 0,Y 632.839,Z 342.393,A -85,B 0,C 180,E1 -5386.726,E2 -5386.726} C_VEL
LIN {X 0,Y 632.842,Z 342.397,A -85,B 0,C 180,E1 -5389.531,E2 -5389.531} C_VEL
LIN {X 0,Y 632.846,Z 342.395,A -85,B 0,C 180,E1 -5392.738,E2 -5392.738} C_VEL
LIN {X 0,Y 632.836,Z 342.394,A -85,B 0,C 180,E1 -5395.56,E2 -5395.56} C_VEL
LIN {X 0,Y 632.856,Z 342.388,A -85,B 0,C 180,E1 -5398.733,E2 -5398.733} C_VEL
LIN {X 0,Y 632.83,Z 342.399,A -85,B 0,C 180,E1 -5401.539,E2 -5401.539} C_VEL
LIN {X 0,Y 632.88,Z 342.396,A -85,B 0,C 180,E1 -5404.622,E2 -5404.622} C_VEL
LIN {X 0,Y 632.824,Z 342.387,A -85,B 0,C 180,E1 -5407.536,E2 -5407.536} C_VEL
LIN {X 0,Y 632.891,Z 342.385,A -85,B 0,C 180,E1 -5410.56,E2 -5410.56} C_VEL
LIN {X 0,Y 632.825,Z 342.398,A -85,B 0,C 180,E1 -5413.524,E2 -5413.524} C_VEL
LIN {X 0,Y 632.893,Z 342.391,A -85,B 0,C 180,E1 -5416.522,E2 -5416.522} C_VEL
LIN {X 0,Y 632.823,Z 342.386,A -85,B 0,C 180,E1 -5419.571,E2 -5419.571} C_VEL
LIN {X 0,Y 632.9,Z 342.387,A -85,B 0,C 180,E1 -5422.576,E2 -5422.576} C_VEL
LIN {X 0,Y 632.825,Z 342.398,A -85,B 0,C 180,E1 -5425.654,E2 -5425.654} C_VEL
LIN {X 0,Y 632.888,Z 342.398,A -85,B 0,C 180,E1 -5428.601,E2 -5428.601} C_VEL
LIN {X 0,Y 632.827,Z 342.398,A -85,B 0,C 180,E1 -5431.64,E2 -5431.64} C_VEL
LIN {X 0,Y 632.855,Z 342.402,A -85,B 0,C 180,E1 -5434.446,E2 -5434.446} C_VEL
LIN {X 0,Y 632.837,Z 342.397,A -85,B 0,C 180,E1 -5437.581,E2 -5437.581} C_VEL
LIN {X 0,Y 632.84,Z 342.403,A -85,B 0,C 180,E1 -5440.376,E2 -5440.376} C_VEL
LIN {X 0,Y 632.839,Z 342.399,A -85,B 0,C 180,E1 -5443.667,E2 -5443.667} C_VEL
LIN {X 0,Y 632.852,Z 342.489,A -85,B 0,C 180,E1 -5446.506,E2 -5446.506} C_VEL
LIN {X 0,Y 641.382,Z 364.278,A -85,B 0,C 180,E1 -5449.122,E2 -5449.122} C_VEL
LIN {X 0,Y 645.735,Z 375.741,A -85,B 0,C 180,E1 -5450.386,E2 -5450.386} C_VEL
LIN {X 0,Y 649.816,Z 383.299,A -85,B 0,C 180,E1 -5450.791,E2 -5450.791} C_VEL
LIN {X 0,Y 655.153,Z 406.516,A -85,B 0,C 180,E1 -5451.491,E2 -5451.491} C_VEL
LIN {X 0,Y 651.371,Z 674.228,A -85,B 0,C 180,E1 -5454.838,E2 -5454.838} C_VEL
LIN {X 0,Y 650.015,Z 767.474,A -85,B 0,C 180,E1 -5456.009,E2 -5456.009} C_VEL
LIN {X 0,Y 649.153,Z 792.825,A -85,B 0,C 180,E1 -5456.482,E2 -5456.482} C_VEL
LIN {X 0,Y 648.242,Z 813.064,A -85,B 0,C 180,E1 -5456.987,E2 -5456.987} C_VEL
LIN {X 0,Y 647.093,Z 835.946,A -85,B 0,C 180,E1 -5457.697,E2 -5457.697} C_VEL
LIN {X 0,Y 645.644,Z 858.657,A -85,B 0,C 180,E1 -5458.575,E2 -5458.575} C_VEL
LIN {X 0,Y 644.282,Z 880.095,A -85,B 0,C 180,E1 -5459.555,E2 -5459.555} C_VEL
LIN {X 0,Y 642.66,Z 902.269,A -85,B 0,C 180,E1 -5460.755,E2 -5460.755} C_VEL
LIN {X 0,Y 641.294,Z 919.982,A -85,B 0,C 180,E1 -5461.859,E2 -5461.859} C_VEL
LIN {X 0,Y 639.606,Z 941.565,A -85,B 0,C 180,E1 -5463.407,E2 -5463.407} C_VEL
LIN {X 0,Y 638.282,Z 958.285,A -85,B 0,C 180,E1 -5464.78,E2 -5464.78} C_VEL
LIN {X 0,Y 636.866,Z 976.749,A -85,B 0,C 180,E1 -5466.498,E2 -5466.498} C_VEL
LIN {X 0,Y 635.732,Z 991.986,A -85,B 0,C 180,E1 -5468.12,E2 -5468.12} C_VEL
LIN {X 0,Y 634.663,Z 1007.703,A -85,B 0,C 180,E1 -5470.009,E2 -5470.009} C_VEL
LIN {X 0,Y 633.812,Z 1021.246,A -85,B 0,C 180,E1 -5471.894,E2 -5471.894} C_VEL
LIN {X 0,Y 633.141,Z 1034.211,A -85,B 0,C 180,E1 -5473.956,E2 -5473.956} C_VEL
LIN {X 0,Y 632.653,Z 1044.642,A -85,B 0,C 180,E1 -5475.913,E2 -5475.913} C_VEL
LIN {X 0,Y 632.316,Z 1053.991,A -85,B 0,C 180,E1 -5477.952,E2 -5477.952} C_VEL
LIN {X 0,Y 632.086,Z 1061.907,A -85,B 0,C 180,E1 -5480.071,E2 -5480.071} C_VEL
LIN {X 0,Y 631.983,Z 1067.745,A -85,B 0,C 180,E1 -5481.997,E2 -5481.997} C_VEL
LIN {X 0,Y 631.933,Z 1073.016,A -85,B 0,C 180,E1 -5484.279,E2 -5484.279} C_VEL
LIN {X 0,Y 631.906,Z 1076.124,A -85,B 0,C 180,E1 -5486.28,E2 -5486.28} C_VEL
LIN {X 0,Y 631.896,Z 1077.969,A -85,B 0,C 180,E1 -5488.277,E2 -5488.277} C_VEL
LIN {X 0,Y 631.893,Z 1078.395,A -85,B 0,C 180,E1 -5490.453,E2 -5490.453} C_VEL
LIN {X 0,Y 631.909,Z 1077.428,A -85,B 0,C 180,E1 -5492.449,E2 -5492.449} C_VEL
LIN {X 0,Y 631.922,Z 1074.768,A -85,B 0,C 180,E1 -5494.72,E2 -5494.72} C_VEL
LIN {X 0,Y 631.937,Z 1070.896,A -85,B 0,C 180,E1 -5496.724,E2 -5496.724} C_VEL
LIN {X 0,Y 632.01,Z 1065.71,A -85,B 0,C 180,E1 -5498.736,E2 -5498.736} C_VEL
LIN {X 0,Y 632.188,Z 1058.309,A -85,B 0,C 180,E1 -5500.941,E2 -5500.941} C_VEL
LIN {X 0,Y 632.439,Z 1050.346,A -85,B 0,C 180,E1 -5502.881,E2 -5502.881} C_VEL
LIN {X 0,Y 632.886,Z 1039.247,A -85,B 0,C 180,E1 -5505.134,E2 -5505.134} C_VEL
LIN {X 0,Y 633.408,Z 1028.544,A -85,B 0,C 180,E1 -5506.98,E2 -5506.98} C_VEL
LIN {X 0,Y 634.203,Z 1014.721,A -85,B 0,C 180,E1 -5509.048,E2 -5509.048} C_VEL
LIN {X 0,Y 635.122,Z 1000.847,A -85,B 0,C 180,E1 -5510.842,E2 -5510.842} C_VEL
LIN {X 0,Y 636.308,Z 984.156,A -85,B 0,C 180,E1 -5512.741,E2 -5512.741} C_VEL
LIN {X 0,Y 637.505,Z 968.256,A -85,B 0,C 180,E1 -5514.319,E2 -5514.319} C_VEL
LIN {X 0,Y 638.959,Z 949.758,A -85,B 0,C 180,E1 -5515.948,E2 -5515.948} C_VEL
LIN {X 0,Y 640.432,Z 931.059,A -85,B 0,C 180,E1 -5517.374,E2 -5517.374} C_VEL
LIN {X 0,Y 642.048,Z 910.744,A -85,B 0,C 180,E1 -5518.742,E2 -5518.742} C_VEL
LIN {X 0,Y 643.519,Z 890.231,A -85,B 0,C 180,E1 -5519.918,E2 -5519.918} C_VEL
LIN {X 0,Y 644.949,Z 869.999,A -85,B 0,C 180,E1 -5520.926,E2 -5520.926} C_VEL
LIN {X 0,Y 646.408,Z 847.179,A -85,B 0,C 180,E1 -5521.887,E2 -5521.887} C_VEL
LIN {X 0,Y 647.553,Z 826.623,A -85,B 0,C 180,E1 -5522.608,E2 -5522.608} C_VEL
LIN {X 0,Y 648.715,Z 803.161,A -85,B 0,C 180,E1 -5523.283,E2 -5523.283} C_VEL
LIN {X 0,Y 649.634,Z 779.407,A -85,B 0,C 180,E1 -5523.789,E2 -5523.789} C_VEL
LIN {X 0,Y 650.311,Z 754.76,A -85,B 0,C 180,E1 -5524.17,E2 -5524.17} C_VEL
LIN {X 0,Y 653.692,Z 505.738,A -85,B 0,C 180,E1 -5527.26,E2 -5527.26} C_VEL
LIN {X 0,Y 654.989,Z 404.942,A -85,B 0,C 180,E1 -5528.542,E2 -5528.542} C_VEL
LIN {X 0,Y 649.257,Z 381.898,A -85,B 0,C 180,E1 -5529.262,E2 -5529.262} C_VEL
LIN {X 0,Y 645.352,Z 374.901,A -85,B 0,C 180,E1 -5529.668,E2 -5529.668} C_VEL
LIN {X 0,Y 637.667,Z 355.005,A -85,B 0,C 180,E1 -5531.912,E2 -5531.912} C_VEL
LIN {X 0,Y 632.849,Z 342.404,A -85,B 0,C 180,E1 -5533.416,E2 -5533.416} C_VEL
LIN {X 0,Y 632.833,Z 342.402,A -85,B 0,C 180,E1 -5536.226,E2 -5536.226} C_VEL
LIN {X 0,Y 632.861,Z 342.395,A -85,B 0,C 180,E1 -5539.387,E2 -5539.387} C_VEL
LIN {X 0,Y 632.826,Z 342.397,A -85,B 0,C 180,E1 -5542.189,E2 -5542.189} C_VEL
LIN {X 0,Y 632.888,Z 342.39,A -85,B 0,C 180,E1 -5545.239,E2 -5545.239} C_VEL
LIN {X 0,Y 632.824,Z 342.395,A -85,B 0,C 180,E1 -5548.219,E2 -5548.219} C_VEL
LIN {X 0,Y 632.902,Z 342.395,A -85,B 0,C 180,E1 -5551.261,E2 -5551.261} C_VEL
LIN {X 0,Y 632.826,Z 342.398,A -85,B 0,C 180,E1 -5554.246,E2 -5554.246} C_VEL
LIN {X 0,Y 632.896,Z 342.382,A -85,B 0,C 180,E1 -5557.228,E2 -5557.228} C_VEL
LIN {X 0,Y 632.825,Z 342.391,A -85,B 0,C 180,E1 -5560.237,E2 -5560.237} C_VEL
LIN {X 0,Y 632.882,Z 342.394,A -85,B 0,C 180,E1 -5563.195,E2 -5563.195} C_VEL
LIN {X 0,Y 632.828,Z 342.394,A -85,B 0,C 180,E1 -5566.29,E2 -5566.29} C_VEL
LIN {X 0,Y 632.866,Z 342.395,A -85,B 0,C 180,E1 -5569.163,E2 -5569.163} C_VEL
LIN {X 0,Y 632.832,Z 342.4,A -85,B 0,C 180,E1 -5572.282,E2 -5572.282} C_VEL
LIN {X 0,Y 632.849,Z 342.388,A -85,B 0,C 180,E1 -5575.106,E2 -5575.106} C_VEL
LIN {X 0,Y 632.841,Z 342.399,A -85,B 0,C 180,E1 -5578.28,E2 -5578.28} C_VEL
LIN {X 0,Y 632.838,Z 342.381,A -85,B 0,C 180,E1 -5581.086,E2 -5581.086} C_VEL
LIN {X 0,Y 632.844,Z 342.394,A -85,B 0,C 180,E1 -5584.35,E2 -5584.35} C_VEL
LIN {X 0,Y 632.838,Z 342.39,A -85,B 0,C 180,E1 -5587.17,E2 -5587.17} C_VEL
LIN {X 0,Y 632.85,Z 342.386,A -85,B 0,C 180,E1 -5590.377,E2 -5590.377} C_VEL
LIN {X 0,Y 632.84,Z 342.396,A -85,B 0,C 180,E1 -5593.274,E2 -5593.274} C_VEL
LIN {X 0,Y 632.847,Z 342.39,A -85,B 0,C 180,E1 -5596.523,E2 -5596.523} C_VEL
LIN {X 0,Y 632.843,Z 342.395,A -85,B 0,C 180,E1 -5599.394,E2 -5599.394} C_VEL
LIN {X 0,Y 632.846,Z 342.4,A -85,B 0,C 180,E1 -5602.676,E2 -5602.676} C_VEL
LIN {X 0,Y 632.836,Z 342.384,A -85,B 0,C 180,E1 -5605.453,E2 -5605.453} C_VEL
LIN {X 0,Y 632.861,Z 342.39,A -85,B 0,C 180,E1 -5608.602,E2 -5608.602} C_VEL
LIN {X 0,Y 632.834,Z 342.398,A -85,B 0,C 180,E1 -5611.438,E2 -5611.438} C_VEL
LIN {X 0,Y 632.879,Z 342.396,A -85,B 0,C 180,E1 -5614.555,E2 -5614.555} C_VEL
LIN {X 0,Y 632.833,Z 342.396,A -85,B 0,C 180,E1 -5617.517,E2 -5617.517} C_VEL
LIN {X 0,Y 632.887,Z 342.393,A -85,B 0,C 180,E1 -5620.611,E2 -5620.611} C_VEL
LIN {X 0,Y 632.83,Z 342.374,A -85,B 0,C 180,E1 -5623.543,E2 -5623.543} C_VEL
LIN {X 0,Y 632.892,Z 342.399,A -85,B 0,C 180,E1 -5626.614,E2 -5626.614} C_VEL
LIN {X 0,Y 632.899,Z 342.393,A -85,B 0,C 180,E1 -5628.635,E2 -5628.635} C_VEL
LIN {X 0,Y 631.782,Z 342.539,A -85,B 0,C 180,E1 -5629.122,E2 -5629.122} C_VEL
LIN {X 0,Y 627.397,Z 343.543,A -85,B 0,C 180,E1 -5629.96,E2 -5629.96} C_VEL
LIN {X 0,Y 625.956,Z 345.103,A -85,B 0,C 180,E1 -5630.399,E2 -5630.399} C_VEL
LIN {X 0,Y 626.203,Z 346.794,A -85,B 0,C 180,E1 -5630.694,E2 -5630.694} C_VEL
LIN {X 0,Y 627.539,Z 350.222,A -85,B 0,C 180,E1 -5631.092,E2 -5631.092} C_VEL
LIN {X 0,Y 646.136,Z 380.402,A -85,B 0,C 180,E1 -5632.915,E2 -5632.915} C_VEL
LIN {X 0,Y 648.908,Z 385.733,A -85,B 0,C 180,E1 -5633.187,E2 -5633.187} C_VEL
LIN {X 0,Y 645.238,Z 625.022,A -85,B 0,C 180,E1 -5636.217,E2 -5636.217} C_VEL
LIN {X 0,Y 643.473,Z 738.636,A -85,B 0,C 180,E1 -5637.656,E2 -5637.656} C_VEL
LIN {X 0,Y 642.583,Z 763.969,A -85,B 0,C 180,E1 -5638.134,E2 -5638.134} C_VEL
LIN {X 0,Y 641.625,Z 784.112,A -85,B 0,C 180,E1 -5638.643,E2 -5638.643} C_VEL
LIN {X 0,Y 640.412,Z 806.612,A -85,B 0,C 180,E1 -5639.35,E2 -5639.35} C_VEL
LIN {X 0,Y 638.823,Z 829.621,A -85,B 0,C 180,E1 -5640.253,E2 -5640.253} C_VEL
LIN {X 0,Y 637.27,Z 851.88,A -85,B 0,C 180,E1 -5641.293,E2 -5641.293} C_VEL
LIN {X 0,Y 635.566,Z 872.666,A -85,B 0,C 180,E1 -5642.45,E2 -5642.45} C_VEL
LIN {X 0,Y 633.988,Z 891.348,A -85,B 0,C 180,E1 -5643.638,E2 -5643.638} C_VEL
LIN {X 0,Y 632.189,Z 912.224,A -85,B 0,C 180,E1 -5645.17,E2 -5645.17} C_VEL
LIN {X 0,Y 630.789,Z 928.845,A -85,B 0,C 180,E1 -5646.555,E2 -5646.555} C_VEL
LIN {X 0,Y 629.177,Z 948.129,A -85,B 0,C 180,E1 -5648.386,E2 -5648.386} C_VEL
LIN {X 0,Y 628.015,Z 962.844,A -85,B 0,C 180,E1 -5649.982,E2 -5649.982} C_VEL
LIN {X 0,Y 626.82,Z 979.01,A -85,B 0,C 180,E1 -5651.973,E2 -5651.973} C_VEL
LIN {X 0,Y 625.963,Z 991.667,A -85,B 0,C 180,E1 -5653.767,E2 -5653.767} C_VEL
LIN {X 0,Y 625.239,Z 1004.457,A -85,B 0,C 180,E1 -5655.837,E2 -5655.837} C_VEL
LIN {X 0,Y 624.721,Z 1014.778,A -85,B 0,C 180,E1 -5657.803,E2 -5657.803} C_VEL
LIN {X 0,Y 624.35,Z 1024.445,A -85,B 0,C 180,E1 -5659.947,E2 -5659.947} C_VEL
LIN {X 0,Y 624.101,Z 1032.207,A -85,B 0,C 180,E1 -5662.08,E2 -5662.08} C_VEL
LIN {X 0,Y 623.99,Z 1037.972,A -85,B 0,C 180,E1 -5664.021,E2 -5664.021} C_VEL
LIN {X 0,Y 623.927,Z 1043.144,A -85,B 0,C 180,E1 -5666.325,E2 -5666.325} C_VEL
LIN {X 0,Y 623.914,Z 1046.095,A -85,B 0,C 180,E1 -5668.255,E2 -5668.255} C_VEL
LIN {X 0,Y 623.9,Z 1048.018,A -85,B 0,C 180,E1 -5670.367,E2 -5670.367} C_VEL
LIN {X 0,Y 623.893,Z 1048.378,A -85,B 0,C 180,E1 -5672.572,E2 -5672.572} C_VEL
LIN {X 0,Y 623.903,Z 1047.444,A -85,B 0,C 180,E1 -5674.504,E2 -5674.504} C_VEL
LIN {X 0,Y 623.921,Z 1044.954,A -85,B 0,C 180,E1 -5676.718,E2 -5676.718} C_VEL
LIN {X 0,Y 623.947,Z 1041.117,A -85,B 0,C 180,E1 -5678.757,E2 -5678.757} C_VEL
LIN {X 0,Y 624.013,Z 1036.208,A -85,B 0,C 180,E1 -5680.712,E2 -5680.712} C_VEL
LIN {X 0,Y 624.202,Z 1028.589,A -85,B 0,C 180,E1 -5683.054,E2 -5683.054} C_VEL
LIN {X 0,Y 624.469,Z 1021.007,A -85,B 0,C 180,E1 -5684.939,E2 -5684.939} C_VEL
LIN {X 0,Y 624.907,Z 1011.141,A -85,B 0,C 180,E1 -5687.026,E2 -5687.026} C_VEL
LIN {X 0,Y 625.479,Z 999.818,A -85,B 0,C 180,E1 -5689.033,E2 -5689.033} C_VEL
LIN {X 0,Y 626.249,Z 987.436,A -85,B 0,C 180,E1 -5690.956,E2 -5690.956} C_VEL
LIN {X 0,Y 627.252,Z 972.986,A -85,B 0,C 180,E1 -5692.89,E2 -5692.89} C_VEL
LIN {X 0,Y 628.31,Z 959.029,A -85,B 0,C 180,E1 -5694.542,E2 -5694.542} C_VEL
LIN {X 0,Y 629.781,Z 940.775,A -85,B 0,C 180,E1 -5696.433,E2 -5696.433} C_VEL
LIN {X 0,Y 631.144,Z 924.5,A -85,B 0,C 180,E1 -5697.914,E2 -5697.914} C_VEL
LIN {X 0,Y 632.941,Z 903.55,A -85,B 0,C 180,E1 -5699.582,E2 -5699.582} C_VEL
LIN {X 0,Y 634.459,Z 885.961,A -85,B 0,C 180,E1 -5700.81,E2 -5700.81} C_VEL
LIN {X 0,Y 636.216,Z 864.814,A -85,B 0,C 180,E1 -5702.101,E2 -5702.101} C_VEL
LIN {X 0,Y 637.795,Z 844.222,A -85,B 0,C 180,E1 -5703.171,E2 -5703.171} C_VEL
LIN {X 0,Y 639.412,Z 822.204,A -85,B 0,C 180,E1 -5704.152,E2 -5704.152} C_VEL
LIN {X 0,Y 640.78,Z 799.713,A -85,B 0,C 180,E1 -5704.969,E2 -5704.969} C_VEL
LIN {X 0,Y 641.872,Z 779.385,A -85,B 0,C 180,E1 -5705.579,E2 -5705.579} C_VEL
LIN {X 0,Y 642.964,Z 753.407,A -85,B 0,C 180,E1 -5706.178,E2 -5706.178} C_VEL
LIN {X 0,Y 643.64,Z 731.33,A -85,B 0,C 180,E1 -5706.539,E2 -5706.539} C_VEL
LIN {X 0,Y 647.419,Z 481.974,A -85,B 0,C 180,E1 -5709.676,E2 -5709.676} C_VEL
LIN {X 0,Y 648.81,Z 385.091,A -85,B 0,C 180,E1 -5710.924,E2 -5710.924} C_VEL
LIN {X 0,Y 635.612,Z 362.835,A -85,B 0,C 180,E1 -5712.239,E2 -5712.239} C_VEL
LIN {X 0,Y 627.277,Z 349.758,A -85,B 0,C 180,E1 -5713.108,E2 -5713.108} C_VEL
LIN {X 0,Y 624.924,Z 343.385,A -85,B 0,C 180,E1 -5713.944,E2 -5713.944} C_VEL
LIN {X 0,Y 624.899,Z 343.386,A -85,B 0,C 180,E1 -5716.856,E2 -5716.856} C_VEL
LIN {X 0,Y 624.916,Z 343.365,A -85,B 0,C 180,E1 -5720.087,E2 -5720.087} C_VEL
LIN {X 0,Y 624.894,Z 343.377,A -85,B 0,C 180,E1 -5722.898,E2 -5722.898} C_VEL
LIN {X 0,Y 624.935,Z 343.381,A -85,B 0,C 180,E1 -5726.055,E2 -5726.055} C_VEL
LIN {X 0,Y 624.893,Z 343.381,A -85,B 0,C 180,E1 -5728.987,E2 -5728.987} C_VEL
LIN {X 0,Y 624.949,Z 343.381,A -85,B 0,C 180,E1 -5732.044,E2 -5732.044} C_VEL
LIN {X 0,Y 624.891,Z 343.38,A -85,B 0,C 180,E1 -5735.012,E2 -5735.012} C_VEL
LIN {X 0,Y 624.949,Z 343.374,A -85,B 0,C 180,E1 -5738.121,E2 -5738.121} C_VEL
LIN {X 0,Y 624.89,Z 343.387,A -85,B 0,C 180,E1 -5741.045,E2 -5741.045} C_VEL
LIN {X 0,Y 624.958,Z 343.383,A -85,B 0,C 180,E1 -5744.122,E2 -5744.122} C_VEL
LIN {X 0,Y 624.888,Z 343.383,A -85,B 0,C 180,E1 -5747.055,E2 -5747.055} C_VEL
LIN {X 0,Y 624.952,Z 343.375,A -85,B 0,C 180,E1 -5750.05,E2 -5750.05} C_VEL
LIN {X 0,Y 624.889,Z 343.385,A -85,B 0,C 180,E1 -5753.107,E2 -5753.107} C_VEL
LIN {X 0,Y 624.952,Z 343.388,A -85,B 0,C 180,E1 -5756.147,E2 -5756.147} C_VEL
LIN {X 0,Y 624.887,Z 343.379,A -85,B 0,C 180,E1 -5759.175,E2 -5759.175} C_VEL
LIN {X 0,Y 624.942,Z 343.379,A -85,B 0,C 180,E1 -5762.109,E2 -5762.109} C_VEL
LIN {X 0,Y 624.89,Z 343.387,A -85,B 0,C 180,E1 -5765.233,E2 -5765.233} C_VEL
LIN {X 0,Y 624.926,Z 343.378,A -85,B 0,C 180,E1 -5768.094,E2 -5768.094} C_VEL
LIN {X 0,Y 624.891,Z 343.374,A -85,B 0,C 180,E1 -5771.257,E2 -5771.257} C_VEL
LIN {X 0,Y 624.924,Z 343.388,A -85,B 0,C 180,E1 -5774.17,E2 -5774.17} C_VEL
LIN {X 0,Y 624.895,Z 343.386,A -85,B 0,C 180,E1 -5777.315,E2 -5777.315} C_VEL
LIN {X 0,Y 624.916,Z 343.377,A -85,B 0,C 180,E1 -5780.219,E2 -5780.219} C_VEL
LIN {X 0,Y 624.896,Z 343.376,A -85,B 0,C 180,E1 -5783.38,E2 -5783.38} C_VEL
LIN {X 0,Y 624.908,Z 343.387,A -85,B 0,C 180,E1 -5786.207,E2 -5786.207} C_VEL
LIN {X 0,Y 624.901,Z 343.385,A -85,B 0,C 180,E1 -5789.421,E2 -5789.421} C_VEL
LIN {X 0,Y 624.898,Z 343.39,A -85,B 0,C 180,E1 -5792.197,E2 -5792.197} C_VEL
LIN {X 0,Y 624.905,Z 343.388,A -85,B 0,C 180,E1 -5795.469,E2 -5795.469} C_VEL
LIN {X 0,Y 624.896,Z 343.389,A -85,B 0,C 180,E1 -5798.261,E2 -5798.261} C_VEL
LIN {X 0,Y 624.91,Z 343.387,A -85,B 0,C 180,E1 -5801.511,E2 -5801.511} C_VEL
LIN {X 0,Y 624.895,Z 343.39,A -85,B 0,C 180,E1 -5804.366,E2 -5804.366} C_VEL
LIN {X 0,Y 624.917,Z 343.598,A -85,B 0,C 180,E1 -5805.924,E2 -5805.924} C_VEL
LIN {X 0,Y 633.318,Z 364.488,A -85,B 0,C 180,E1 -5808.517,E2 -5808.517} C_VEL
LIN {X 0,Y 637.458,Z 375.458,A -85,B 0,C 180,E1 -5809.756,E2 -5809.756} C_VEL
LIN {X 0,Y 644.114,Z 387.269,A -85,B 0,C 180,E1 -5810.43,E2 -5810.43} C_VEL
LIN {X 0,Y 648.865,Z 408.283,A -85,B 0,C 180,E1 -5811.072,E2 -5811.072} C_VEL
LIN {X 0,Y 644.789,Z 676.123,A -85,B 0,C 180,E1 -5814.454,E2 -5814.454} C_VEL
LIN {X 0,Y 643.359,Z 767.457,A -85,B 0,C 180,E1 -5815.612,E2 -5815.612} C_VEL
LIN {X 0,Y 642.441,Z 792.729,A -85,B 0,C 180,E1 -5816.088,E2 -5816.088} C_VEL
LIN {X 0,Y 641.474,Z 812.839,A -85,B 0,C 180,E1 -5816.594,E2 -5816.594} C_VEL
LIN {X 0,Y 640.273,Z 835.294,A -85,B 0,C 180,E1 -5817.294,E2 -5817.294} C_VEL
LIN {X 0,Y 638.713,Z 858.184,A -85,B 0,C 180,E1 -5818.183,E2 -5818.183} C_VEL
LIN {X 0,Y 637.286,Z 878.858,A -85,B 0,C 180,E1 -5819.132,E2 -5819.132} C_VEL
LIN {X 0,Y 635.566,Z 901.227,A -85,B 0,C 180,E1 -5820.345,E2 -5820.345} C_VEL
LIN {X 0,Y 634.055,Z 919.856,A -85,B 0,C 180,E1 -5821.508,E2 -5821.508} C_VEL
LIN {X 0,Y 632.282,Z 941.134,A -85,B 0,C 180,E1 -5823.038,E2 -5823.038} C_VEL
LIN {X 0,Y 630.831,Z 958.283,A -85,B 0,C 180,E1 -5824.461,E2 -5824.461} C_VEL
LIN {X 0,Y 629.293,Z 976.747,A -85,B 0,C 180,E1 -5826.198,E2 -5826.198} C_VEL
LIN {X 0,Y 628.078,Z 991.933,A -85,B 0,C 180,E1 -5827.833,E2 -5827.833} C_VEL
LIN {X 0,Y 626.909,Z 1007.705,A -85,B 0,C 180,E1 -5829.751,E2 -5829.751} C_VEL
LIN {X 0,Y 625.997,Z 1021.244,A -85,B 0,C 180,E1 -5831.659,E2 -5831.659} C_VEL
LIN {X 0,Y 625.286,Z 1033.689,A -85,B 0,C 180,E1 -5833.654,E2 -5833.654} C_VEL
LIN {X 0,Y 624.723,Z 1044.641,A -85,B 0,C 180,E1 -5835.731,E2 -5835.731} C_VEL
LIN {X 0,Y 624.367,Z 1053.585,A -85,B 0,C 180,E1 -5837.702,E2 -5837.702} C_VEL
LIN {X 0,Y 624.106,Z 1061.907,A -85,B 0,C 180,E1 -5839.943,E2 -5839.943} C_VEL
LIN {X 0,Y 624.01,Z 1067.49,A -85,B 0,C 180,E1 -5841.801,E2 -5841.801} C_VEL
LIN {X 0,Y 623.94,Z 1072.696,A -85,B 0,C 180,E1 -5844.021,E2 -5844.021} C_VEL
LIN {X 0,Y 623.907,Z 1076.01,A -85,B 0,C 180,E1 -5846.14,E2 -5846.14} C_VEL
LIN {X 0,Y 623.904,Z 1077.836,A -85,B 0,C 180,E1 -5848.071,E2 -5848.071} C_VEL
LIN {X 0,Y 623.895,Z 1078.417,A -85,B 0,C 180,E1 -5850.367,E2 -5850.367} C_VEL
LIN {X 0,Y 623.91,Z 1077.496,A -85,B 0,C 180,E1 -5852.388,E2 -5852.388} C_VEL
LIN {X 0,Y 623.919,Z 1075.085,A -85,B 0,C 180,E1 -5854.596,E2 -5854.596} C_VEL
LIN {X 0,Y 623.939,Z 1071.102,A -85,B 0,C 180,E1 -5856.718,E2 -5856.718} C_VEL
LIN {X 0,Y 624.014,Z 1066.219,A -85,B 0,C 180,E1 -5858.663,E2 -5858.663} C_VEL
LIN {X 0,Y 624.206,Z 1058.661,A -85,B 0,C 180,E1 -5860.989,E2 -5860.989} C_VEL
LIN {X 0,Y 624.476,Z 1050.75,A -85,B 0,C 180,E1 -5862.954,E2 -5862.954} C_VEL
LIN {X 0,Y 624.93,Z 1040.405,A -85,B 0,C 180,E1 -5865.118,E2 -5865.118} C_VEL
LIN {X 0,Y 625.518,Z 1029.116,A -85,B 0,C 180,E1 -5867.105,E2 -5867.105} C_VEL
LIN {X 0,Y 626.333,Z 1016.12,A -85,B 0,C 180,E1 -5869.103,E2 -5869.103} C_VEL
LIN {X 0,Y 627.354,Z 1001.616,A -85,B 0,C 180,E1 -5871.015,E2 -5871.015} C_VEL
LIN {X 0,Y 628.562,Z 986,A -85,B 0,C 180,E1 -5872.839,E2 -5872.839} C_VEL
LIN {X 0,Y 629.943,Z 968.823,A -85,B 0,C 180,E1 -5874.574,E2 -5874.574} C_VEL
LIN {X 0,Y 631.502,Z 950.498,A -85,B 0,C 180,E1 -5876.216,E2 -5876.216} C_VEL
LIN {X 0,Y 633.079,Z 931.694,A -85,B 0,C 180,E1 -5877.668,E2 -5877.668} C_VEL
LIN {X 0,Y 634.609,Z 913.191,A -85,B 0,C 180,E1 -5878.928,E2 -5878.928} C_VEL
LIN {X 0,Y 636.354,Z 890.919,A -85,B 0,C 180,E1 -5880.238,E2 -5880.238} C_VEL
LIN {X 0,Y 637.792,Z 871.802,A -85,B 0,C 180,E1 -5881.207,E2 -5881.207} C_VEL
LIN {X 0,Y 639.438,Z 848.234,A -85,B 0,C 180,E1 -5882.224,E2 -5882.224} C_VEL
LIN {X 0,Y 640.692,Z 827.149,A -85,B 0,C 180,E1 -5882.975,E2 -5882.975} C_VEL
LIN {X 0,Y 641.942,Z 803.825,A -85,B 0,C 180,E1 -5883.657,E2 -5883.657} C_VEL
LIN {X 0,Y 642.944,Z 779.718,A -85,B 0,C 180,E1 -5884.178,E2 -5884.178} C_VEL
LIN {X 0,Y 643.646,Z 755.972,A -85,B 0,C 180,E1 -5884.552,E2 -5884.552} C_VEL
LIN {X 0,Y 647.272,Z 508.069,A -85,B 0,C 180,E1 -5887.659,E2 -5887.659} C_VEL
LIN {X 0,Y 648.694,Z 406.811,A -85,B 0,C 180,E1 -5888.956,E2 -5888.956} C_VEL
LIN {X 0,Y 643.579,Z 386.076,A -85,B 0,C 180,E1 -5889.609,E2 -5889.609} C_VEL
LIN {X 0,Y 636.999,Z 374.634,A -85,B 0,C 180,E1 -5890.282,E2 -5890.282} C_VEL
LIN {X 0,Y 630.181,Z 356.926,A -85,B 0,C 180,E1 -5892.32,E2 -5892.32} C_VEL
LIN {X 0,Y 625.657,Z 345.944,A -85,B 0,C 180,E1 -5893.662,E2 -5893.662} C_VEL
LIN {X 0,Y 624.887,Z 343.395,A -85,B 0,C 180,E1 -5893.983,E2 -5893.983} C_VEL
LIN {X 0,Y 624.953,Z 343.388,A -85,B 0,C 180,E1 -5897.033,E2 -5897.033} C_VEL
LIN {X 0,Y 624.886,Z 343.382,A -85,B 0,C 180,E1 -5900.037,E2 -5900.037} C_VEL
LIN {X 0,Y 624.956,Z 343.376,A -85,B 0,C 180,E1 -5903.017,E2 -5903.017} C_VEL
LIN {X 0,Y 624.887,Z 343.383,A -85,B 0,C 180,E1 -5906.052,E2 -5906.052} C_VEL
LIN {X 0,Y 624.955,Z 343.374,A -85,B 0,C 180,E1 -5909.097,E2 -5909.097} C_VEL
LIN {X 0,Y 624.889,Z 343.378,A -85,B 0,C 180,E1 -5912.145,E2 -5912.145} C_VEL
LIN {X 0,Y 624.956,Z 343.385,A -85,B 0,C 180,E1 -5915.217,E2 -5915.217} C_VEL
LIN {X 0,Y 624.887,Z 343.388,A -85,B 0,C 180,E1 -5918.209,E2 -5918.209} C_VEL
LIN {X 0,Y 624.939,Z 343.372,A -85,B 0,C 180,E1 -5921.144,E2 -5921.144} C_VEL
LIN {X 0,Y 624.891,Z 343.384,A -85,B 0,C 180,E1 -5924.216,E2 -5924.216} C_VEL
LIN {X 0,Y 624.92,Z 343.379,A -85,B 0,C 180,E1 -5927.056,E2 -5927.056} C_VEL
LIN {X 0,Y 624.894,Z 343.373,A -85,B 0,C 180,E1 -5930.235,E2 -5930.235} C_VEL
LIN {X 0,Y 624.915,Z 343.385,A -85,B 0,C 180,E1 -5933.108,E2 -5933.108} C_VEL
LIN {X 0,Y 624.896,Z 343.383,A -85,B 0,C 180,E1 -5936.33,E2 -5936.33} C_VEL
LIN {X 0,Y 624.912,Z 343.384,A -85,B 0,C 180,E1 -5939.175,E2 -5939.175} C_VEL
LIN {X 0,Y 624.9,Z 343.389,A -85,B 0,C 180,E1 -5942.384,E2 -5942.384} C_VEL
LIN {X 0,Y 624.907,Z 343.379,A -85,B 0,C 180,E1 -5945.233,E2 -5945.233} C_VEL
LIN {X 0,Y 624.903,Z 343.389,A -85,B 0,C 180,E1 -5948.465,E2 -5948.465} C_VEL
LIN {X 0,Y 624.908,Z 343.369,A -85,B 0,C 180,E1 -5951.35,E2 -5951.35} C_VEL
LIN {X 0,Y 624.904,Z 343.384,A -85,B 0,C 180,E1 -5954.549,E2 -5954.549} C_VEL
LIN {X 0,Y 624.907,Z 343.38,A -85,B 0,C 180,E1 -5957.41,E2 -5957.41} C_VEL
LIN {X 0,Y 624.906,Z 343.375,A -85,B 0,C 180,E1 -5960.611,E2 -5960.611} C_VEL
LIN {X 0,Y 624.899,Z 343.386,A -85,B 0,C 180,E1 -5963.38,E2 -5963.38} C_VEL
LIN {X 0,Y 624.918,Z 343.387,A -85,B 0,C 180,E1 -5966.616,E2 -5966.616} C_VEL
LIN {X 0,Y 624.895,Z 343.374,A -85,B 0,C 180,E1 -5969.422,E2 -5969.422} C_VEL
LIN {X 0,Y 624.941,Z 343.379,A -85,B 0,C 180,E1 -5972.522,E2 -5972.522} C_VEL
LIN {X 0,Y 624.896,Z 343.387,A -85,B 0,C 180,E1 -5975.509,E2 -5975.509} C_VEL
LIN {X 0,Y 624.937,Z 343.387,A -85,B 0,C 180,E1 -5978.667,E2 -5978.667} C_VEL
LIN {X 0,Y 624.896,Z 343.391,A -85,B 0,C 180,E1 -5981.609,E2 -5981.609} C_VEL
LIN {X 0,Y 624.934,Z 343.351,A -85,B 0,C 180,E1 -5984.749,E2 -5984.749} C_VEL
LIN {X 0,Y 624.894,Z 343.384,A -85,B 0,C 180,E1 -5987.667,E2 -5987.667} C_VEL
LIN {X 0,Y 624.953,Z 343.473,A -85,B 0,C 180,E1 -5990.27,E2 -5990.27} C_VEL
LIN {X 0,Y 626.203,Z 346.794,A -85,B 0,C 180,E1 -5990.694,E2 -5990.694} C_VEL
LIN {X 0,Y 627.768,Z 350.392,A -85,B 0,C 180,E1 -5991.039,E2 -5991.039} C_VEL
LIN {X 0,Y 629.852,Z 356.916,A -85,B 0,C 180,E1 -5991.369,E2 -5991.369} C_VEL
LIN {X 0,Y 633.845,Z 372.513,A -85,B 0,C 180,E1 -5991.9,E2 -5991.9} C_VEL
LIN {X 0,Y 635.947,Z 377.186,A -85,B 0,C 180,E1 -5992.125,E2 -5992.125} C_VEL
LIN {X 0,Y 642.615,Z 388.681,A -85,B 0,C 180,E1 -5992.777,E2 -5992.777} C_VEL
LIN {X 0,Y 638.708,Z 628.744,A -85,B 0,C 180,E1 -5995.841,E2 -5995.841} C_VEL
LIN {X 0,Y 636.879,Z 738.868,A -85,B 0,C 180,E1 -5997.249,E2 -5997.249} C_VEL
LIN {X 0,Y 635.934,Z 764.323,A -85,B 0,C 180,E1 -5997.734,E2 -5997.734} C_VEL
LIN {X 0,Y 634.929,Z 784.357,A -85,B 0,C 180,E1 -5998.245,E2 -5998.245} C_VEL
LIN {X 0,Y 633.679,Z 806.259,A -85,B 0,C 180,E1 -5998.937,E2 -5998.937} C_VEL
LIN {X 0,Y 631.998,Z 829.361,A -85,B 0,C 180,E1 -5999.846,E2 -5999.846} C_VEL
LIN {X 0,Y 630.445,Z 849.976,A -85,B 0,C 180,E1 -6000.811,E2 -6000.811} C_VEL
LIN {X 0,Y 628.6,Z 871.75,A -85,B 0,C 180,E1 -6002.015,E2 -6002.015} C_VEL
LIN {X 0,Y 626.972,Z 889.893,A -85,B 0,C 180,E1 -6003.171,E2 -6003.171} C_VEL
LIN {X 0,Y 625.011,Z 910.955,A -85,B 0,C 180,E1 -6004.713,E2 -6004.713} C_VEL
LIN {X 0,Y 623.503,Z 927.172,A -85,B 0,C 180,E1 -6006.077,E2 -6006.077} C_VEL
LIN {X 0,Y 621.814,Z 945.972,A -85,B 0,C 180,E1 -6007.854,E2 -6007.854} C_VEL
LIN {X 0,Y 620.415,Z 962.253,A -85,B 0,C 180,E1 -6009.628,E2 -6009.628} C_VEL
LIN {X 0,Y 619.163,Z 977.823,A -85,B 0,C 180,E1 -6011.547,E2 -6011.547} C_VEL
LIN {X 0,Y 618.189,Z 991.221,A -85,B 0,C 180,E1 -6013.461,E2 -6013.461} C_VEL
LIN {X 0,Y 617.383,Z 1004.094,A -85,B 0,C 180,E1 -6015.557,E2 -6015.557} C_VEL
LIN {X 0,Y 616.791,Z 1014.91,A -85,B 0,C 180,E1 -6017.644,E2 -6017.644} C_VEL
LIN {X 0,Y 616.386,Z 1024.556,A -85,B 0,C 180,E1 -6019.816,E2 -6019.816} C_VEL
LIN {X 0,Y 616.118,Z 1032.294,A -85,B 0,C 180,E1 -6021.977,E2 -6021.977} C_VEL
LIN {X 0,Y 616.001,Z 1038.045,A -85,B 0,C 180,E1 -6023.944,E2 -6023.944} C_VEL
LIN {X 0,Y 615.93,Z 1043.189,A -85,B 0,C 180,E1 -6026.277,E2 -6026.277} C_VEL
LIN {X 0,Y 615.915,Z 1046.127,A -85,B 0,C 180,E1 -6028.232,E2 -6028.232} C_VEL
LIN {X 0,Y 615.9,Z 1048.037,A -85,B 0,C 180,E1 -6030.372,E2 -6030.372} C_VEL
LIN {X 0,Y 615.894,Z 1048.372,A -85,B 0,C 180,E1 -6032.605,E2 -6032.605} C_VEL
LIN {X 0,Y 615.9,Z 1047.414,A -85,B 0,C 180,E1 -6034.577,E2 -6034.577} C_VEL
LIN {X 0,Y 615.92,Z 1044.749,A -85,B 0,C 180,E1 -6036.9,E2 -6036.9} C_VEL
LIN {X 0,Y 615.961,Z 1040.849,A -85,B 0,C 180,E1 -6038.965,E2 -6038.965} C_VEL
LIN {X 0,Y 616.051,Z 1035.367,A -85,B 0,C 180,E1 -6041.136,E2 -6041.136} C_VEL
LIN {X 0,Y 616.246,Z 1028.13,A -85,B 0,C 180,E1 -6043.321,E2 -6043.321} C_VEL
LIN {X 0,Y 616.539,Z 1020.478,A -85,B 0,C 180,E1 -6045.232,E2 -6045.232} C_VEL
LIN {X 0,Y 617.068,Z 1009.43,A -85,B 0,C 180,E1 -6047.541,E2 -6047.541} C_VEL
LIN {X 0,Y 617.72,Z 998.488,A -85,B 0,C 180,E1 -6049.478,E2 -6049.478} C_VEL
LIN {X 0,Y 618.662,Z 984.485,A -85,B 0,C 180,E1 -6051.623,E2 -6051.623} C_VEL
LIN {X 0,Y 619.676,Z 971.194,A -85,B 0,C 180,E1 -6053.387,E2 -6053.387} C_VEL
LIN {X 0,Y 621.016,Z 955.276,A -85,B 0,C 180,E1 -6055.257,E2 -6055.257} C_VEL
LIN {X 0,Y 622.444,Z 938.805,A -85,B 0,C 180,E1 -6056.937,E2 -6056.937} C_VEL
LIN {X 0,Y 624.226,Z 919.692,A -85,B 0,C 180,E1 -6058.668,E2 -6058.668} C_VEL
LIN {X 0,Y 625.918,Z 901.36,A -85,B 0,C 180,E1 -6060.106,E2 -6060.106} C_VEL
LIN {X 0,Y 627.697,Z 882.047,A -85,B 0,C 180,E1 -6061.446,E2 -6061.446} C_VEL
LIN {X 0,Y 629.506,Z 861.113,A -85,B 0,C 180,E1 -6062.687,E2 -6062.687} C_VEL
LIN {X 0,Y 631.175,Z 840.831,A -85,B 0,C 180,E1 -6063.727,E2 -6063.727} C_VEL
LIN {X 0,Y 632.919,Z 817.134,A -85,B 0,C 180,E1 -6064.744,E2 -6064.744} C_VEL
LIN {X 0,Y 634.242,Z 796.202,A -85,B 0,C 180,E1 -6065.489,E2 -6065.489} C_VEL
LIN {X 0,Y 635.639,Z 770.4,A -85,B 0,C 180,E1 -6066.215,E2 -6066.215} C_VEL
LIN {X 0,Y 636.544,Z 749.103,A -85,B 0,C 180,E1 -6066.666,E2 -6066.666} C_VEL
LIN {X 0,Y 637.275,Z 721.539,A -85,B 0,C 180,E1 -6067.081,E2 -6067.081} C_VEL
LIN {X 0,Y 641.355,Z 468.268,A -85,B 0,C 180,E1 -6070.294,E2 -6070.294} C_VEL
LIN {X 0,Y 642.577,Z 388.154,A -85,B 0,C 180,E1 -6071.34,E2 -6071.34} C_VEL
LIN {X 0,Y 628.337,Z 364.446,A -85,B 0,C 180,E1 -6072.794,E2 -6072.794} C_VEL
LIN {X 0,Y 619.079,Z 350.106,A -85,B 0,C 180,E1 -6073.783,E2 -6073.783} C_VEL
LIN {X 0,Y 616.951,Z 344.375,A -85,B 0,C 180,E1 -6074.568,E2 -6074.568} C_VEL
LIN {X 0,Y 617.017,Z 344.368,A -85,B 0,C 180,E1 -6077.643,E2 -6077.643} C_VEL
LIN {X 0,Y 616.95,Z 344.369,A -85,B 0,C 180,E1 -6080.677,E2 -6080.677} C_VEL
LIN {X 0,Y 617.011,Z 344.339,A -85,B 0,C 180,E1 -6083.736,E2 -6083.736} C_VEL
LIN {X 0,Y 616.951,Z 344.377,A -85,B 0,C 180,E1 -6086.784,E2 -6086.784} C_VEL
LIN {X 0,Y 617.02,Z 344.373,A -85,B 0,C 180,E1 -6089.923,E2 -6089.923} C_VEL
LIN {X 0,Y 616.953,Z 344.377,A -85,B 0,C 180,E1 -6092.908,E2 -6092.908} C_VEL
LIN {X 0,Y 617.012,Z 344.374,A -85,B 0,C 180,E1 -6096.062,E2 -6096.062} C_VEL
LIN {X 0,Y 616.95,Z 344.37,A -85,B 0,C 180,E1 -6099.012,E2 -6099.012} C_VEL
LIN {X 0,Y 617.016,Z 344.363,A -85,B 0,C 180,E1 -6102.067,E2 -6102.067} C_VEL
LIN {X 0,Y 616.95,Z 344.375,A -85,B 0,C 180,E1 -6105.067,E2 -6105.067} C_VEL
LIN {X 0,Y 617.015,Z 344.374,A -85,B 0,C 180,E1 -6108.123,E2 -6108.123} C_VEL
LIN {X 0,Y 616.949,Z 344.372,A -85,B 0,C 180,E1 -6111.143,E2 -6111.143} C_VEL
LIN {X 0,Y 617.016,Z 344.362,A -85,B 0,C 180,E1 -6114.14,E2 -6114.14} C_VEL
LIN {X 0,Y 616.948,Z 344.376,A -85,B 0,C 180,E1 -6117.213,E2 -6117.213} C_VEL
LIN {X 0,Y 617.023,Z 344.375,A -85,B 0,C 180,E1 -6120.279,E2 -6120.279} C_VEL
LIN {X 0,Y 616.947,Z 344.366,A -85,B 0,C 180,E1 -6123.345,E2 -6123.345} C_VEL
LIN {X 0,Y 617.018,Z 344.361,A -85,B 0,C 180,E1 -6126.42,E2 -6126.42} C_VEL
LIN {X 0,Y 616.949,Z 344.376,A -85,B 0,C 180,E1 -6129.421,E2 -6129.421} C_VEL
LIN {X 0,Y 617.014,Z 344.368,A -85,B 0,C 180,E1 -6132.447,E2 -6132.447} C_VEL
LIN {X 0,Y 616.947,Z 344.364,A -85,B 0,C 180,E1 -6135.511,E2 -6135.511} C_VEL
LIN {X 0,Y 617.015,Z 344.364,A -85,B 0,C 180,E1 -6138.557,E2 -6138.557} C_VEL
LIN {X 0,Y 616.948,Z 344.376,A -85,B 0,C 180,E1 -6141.586,E2 -6141.586} C_VEL
LIN {X 0,Y 617.003,Z 344.37,A -85,B 0,C 180,E1 -6144.511,E2 -6144.511} C_VEL
LIN {X 0,Y 616.951,Z 344.371,A -85,B 0,C 180,E1 -6147.615,E2 -6147.615} C_VEL
LIN {X 0,Y 616.989,Z 344.378,A -85,B 0,C 180,E1 -6150.481,E2 -6150.481} C_VEL
LIN {X 0,Y 616.953,Z 344.378,A -85,B 0,C 180,E1 -6153.661,E2 -6153.661} C_VEL
LIN {X 0,Y 616.991,Z 344.377,A -85,B 0,C 180,E1 -6156.611,E2 -6156.611} C_VEL
LIN {X 0,Y 616.956,Z 344.379,A -85,B 0,C 180,E1 -6159.684,E2 -6159.684} C_VEL
LIN {X 0,Y 616.969,Z 344.367,A -85,B 0,C 180,E1 -6162.517,E2 -6162.517} C_VEL
LIN {X 0,Y 617.023,Z 344.531,A -85,B 0,C 180,E1 -6165.308,E2 -6165.308} C_VEL
LIN {X 0,Y 625.556,Z 365.763,A -85,B 0,C 180,E1 -6168.01,E2 -6168.01} C_VEL
LIN {X 0,Y 629.163,Z 375.222,A -85,B 0,C 180,E1 -6169.101,E2 -6169.101} C_VEL
LIN {X 0,Y 638.485,Z 391.346,A -85,B 0,C 180,E1 -6170.065,E2 -6170.065} C_VEL
LIN {X 0,Y 642.629,Z 410.143,A -85,B 0,C 180,E1 -6170.645,E2 -6170.645} C_VEL
LIN {X 0,Y 638.252,Z 676.966,A -85,B 0,C 180,E1 -6174.048,E2 -6174.048} C_VEL
LIN {X 0,Y 636.738,Z 767.252,A -85,B 0,C 180,E1 -6175.203,E2 -6175.203} C_VEL
LIN {X 0,Y 635.766,Z 792.504,A -85,B 0,C 180,E1 -6175.683,E2 -6175.683} C_VEL
LIN {X 0,Y 634.738,Z 812.614,A -85,B 0,C 180,E1 -6176.192,E2 -6176.192} C_VEL
LIN {X 0,Y 633.457,Z 835.069,A -85,B 0,C 180,E1 -6176.897,E2 -6176.897} C_VEL
LIN {X 0,Y 631.844,Z 857.447,A -85,B 0,C 180,E1 -6177.771,E2 -6177.771} C_VEL
LIN {X 0,Y 630.335,Z 877.622,A -85,B 0,C 180,E1 -6178.701,E2 -6178.701} C_VEL
LIN {X 0,Y 628.484,Z 900.405,A -85,B 0,C 180,E1 -6179.938,E2 -6179.938} C_VEL
LIN {X 0,Y 626.885,Z 918.89,A -85,B 0,C 180,E1 -6181.1,E2 -6181.1} C_VEL
LIN {X 0,Y 625.021,Z 939.869,A -85,B 0,C 180,E1 -6182.608,E2 -6182.608} C_VEL
LIN {X 0,Y 623.487,Z 957.138,A -85,B 0,C 180,E1 -6184.036,E2 -6184.036} C_VEL
LIN {X 0,Y 621.967,Z 974.396,A -85,B 0,C 180,E1 -6185.647,E2 -6185.647} C_VEL
LIN {X 0,Y 620.503,Z 991.086,A -85,B 0,C 180,E1 -6187.448,E2 -6187.448} C_VEL
LIN {X 0,Y 619.292,Z 1006.237,A -85,B 0,C 180,E1 -6189.293,E2 -6189.293} C_VEL
LIN {X 0,Y 618.235,Z 1020.607,A -85,B 0,C 180,E1 -6191.323,E2 -6191.323} C_VEL
LIN {X 0,Y 617.432,Z 1033.123,A -85,B 0,C 180,E1 -6193.343,E2 -6193.343} C_VEL
LIN {X 0,Y 616.82,Z 1044.181,A -85,B 0,C 180,E1 -6195.448,E2 -6195.448} C_VEL
LIN {X 0,Y 616.445,Z 1052.774,A -85,B 0,C 180,E1 -6197.351,E2 -6197.351} C_VEL
LIN {X 0,Y 616.144,Z 1061.604,A -85,B 0,C 180,E1 -6199.717,E2 -6199.717} C_VEL
LIN {X 0,Y 616.019,Z 1067.49,A -85,B 0,C 180,E1 -6201.694,E2 -6201.694} C_VEL
LIN {X 0,Y 615.943,Z 1072.696,A -85,B 0,C 180,E1 -6203.943,E2 -6203.943} C_VEL
LIN {X 0,Y 615.908,Z 1076.01,A -85,B 0,C 180,E1 -6206.09,E2 -6206.09} C_VEL
LIN {X 0,Y 615.905,Z 1077.836,A -85,B 0,C 180,E1 -6208.046,E2 -6208.046} C_VEL
LIN {X 0,Y 615.895,Z 1078.417,A -85,B 0,C 180,E1 -6210.372,E2 -6210.372} C_VEL
LIN {X 0,Y 615.909,Z 1077.495,A -85,B 0,C 180,E1 -6212.419,E2 -6212.419} C_VEL
LIN {X 0,Y 615.921,Z 1075.085,A -85,B 0,C 180,E1 -6214.656,E2 -6214.656} C_VEL
LIN {X 0,Y 615.947,Z 1071.102,A -85,B 0,C 180,E1 -6216.806,E2 -6216.806} C_VEL
LIN {X 0,Y 616.023,Z 1066.219,A -85,B 0,C 180,E1 -6218.776,E2 -6218.776} C_VEL
LIN {X 0,Y 616.234,Z 1058.661,A -85,B 0,C 180,E1 -6221.133,E2 -6221.133} C_VEL
LIN {X 0,Y 616.531,Z 1050.749,A -85,B 0,C 180,E1 -6223.124,E2 -6223.124} C_VEL
LIN {X 0,Y 617.024,Z 1040.404,A -85,B 0,C 180,E1 -6225.316,E2 -6225.316} C_VEL
LIN {X 0,Y 617.67,Z 1029.115,A -85,B 0,C 180,E1 -6227.329,E2 -6227.329} C_VEL
LIN {X 0,Y 618.548,Z 1016.119,A -85,B 0,C 180,E1 -6229.353,E2 -6229.353} C_VEL
LIN {X 0,Y 619.65,Z 1001.614,A -85,B 0,C 180,E1 -6231.289,E2 -6231.289} C_VEL
LIN {X 0,Y 620.977,Z 985.782,A -85,B 0,C 180,E1 -6233.158,E2 -6233.158} C_VEL
LIN {X 0,Y 622.442,Z 968.822,A -85,B 0,C 180,E1 -6234.89,E2 -6234.89} C_VEL
LIN {X 0,Y 623.88,Z 952.658,A -85,B 0,C 180,E1 -6236.356,E2 -6236.356} C_VEL
LIN {X 0,Y 625.655,Z 932.82,A -85,B 0,C 180,E1 -6237.921,E2 -6237.921} C_VEL
LIN {X 0,Y 627.208,Z 915.193,A -85,B 0,C 180,E1 -6239.145,E2 -6239.145} C_VEL
LIN {X 0,Y 629.064,Z 893.416,A -85,B 0,C 180,E1 -6240.467,E2 -6240.467} C_VEL
LIN {X 0,Y 630.661,Z 873.465,A -85,B 0,C 180,E1 -6241.501,E2 -6241.501} C_VEL
LIN {X 0,Y 632.318,Z 851.795,A -85,B 0,C 180,E1 -6242.47,E2 -6242.47} C_VEL
LIN {X 0,Y 633.817,Z 828.417,A -85,B 0,C 180,E1 -6243.325,E2 -6243.325} C_VEL
LIN {X 0,Y 635.03,Z 807.166,A -85,B 0,C 180,E1 -6243.962,E2 -6243.962} C_VEL
LIN {X 0,Y 636.216,Z 781.646,A -85,B 0,C 180,E1 -6244.545,E2 -6244.545} C_VEL
LIN {X 0,Y 636.941,Z 759.56,A -85,B 0,C 180,E1 -6244.907,E2 -6244.907} C_VEL
LIN {X 0,Y 640.729,Z 518.976,A -85,B 0,C 180,E1 -6247.955,E2 -6247.955} C_VEL
LIN {X 0,Y 642.4,Z 408.639,A -85,B 0,C 180,E1 -6249.376,E2 -6249.376} C_VEL
LIN {X 0,Y 637.907,Z 390.365,A -85,B 0,C 180,E1 -6249.96,E2 -6249.96} C_VEL
LIN {X 0,Y 628.778,Z 374.728,A -85,B 0,C 180,E1 -6250.874,E2 -6250.874} C_VEL
LIN {X 0,Y 620.891,Z 354.378,A -85,B 0,C 180,E1 -6253.289,E2 -6253.289} C_VEL
LIN {X 0,Y 616.988,Z 344.415,A -85,B 0,C 180,E1 -6254.53,E2 -6254.53} C_VEL
LIN {X 0,Y 616.953,Z 344.382,A -85,B 0,C 180,E1 -6257.733,E2 -6257.733} C_VEL
LIN {X 0,Y 616.974,Z 344.369,A -85,B 0,C 180,E1 -6260.558,E2 -6260.558} C_VEL
LIN {X 0,Y 616.959,Z 344.381,A -85,B 0,C 180,E1 -6263.733,E2 -6263.733} C_VEL
LIN {X 0,Y 616.967,Z 344.37,A -85,B 0,C 180,E1 -6266.578,E2 -6266.578} C_VEL
LIN {X 0,Y 616.959,Z 344.375,A -85,B 0,C 180,E1 -6269.84,E2 -6269.84} C_VEL
LIN {X 0,Y 616.964,Z 344.364,A -85,B 0,C 180,E1 -6272.638,E2 -6272.638} C_VEL
LIN {X 0,Y 616.962,Z 344.366,A -85,B 0,C 180,E1 -6275.895,E2 -6275.895} C_VEL
LIN {X 0,Y 616.964,Z 344.374,A -85,B 0,C 180,E1 -6278.73,E2 -6278.73} C_VEL
LIN {X 0,Y 616.961,Z 344.376,A -85,B 0,C 180,E1 -6282.051,E2 -6282.051} C_VEL
LIN {X 0,Y 616.976,Z 344.369,A -85,B 0,C 180,E1 -6284.971,E2 -6284.971} C_VEL
LIN {X 0,Y 616.957,Z 344.377,A -85,B 0,C 180,E1 -6288.217,E2 -6288.217} C_VEL
LIN {X 0,Y 616.981,Z 344.358,A -85,B 0,C 180,E1 -6291.144,E2 -6291.144} C_VEL
LIN {X 0,Y 616.956,Z 344.369,A -85,B 0,C 180,E1 -6294.326,E2 -6294.326} C_VEL
LIN {X 0,Y 616.99,Z 344.368,A -85,B 0,C 180,E1 -6297.306,E2 -6297.306} C_VEL
LIN {X 0,Y 616.953,Z 344.359,A -85,B 0,C 180,E1 -6300.475,E2 -6300.475} C_VEL
LIN {X 0,Y 616.993,Z 344.373,A -85,B 0,C 180,E1 -6303.438,E2 -6303.438} C_VEL
LIN {X 0,Y 616.952,Z 344.369,A -85,B 0,C 180,E1 -6306.608,E2 -6306.608} C_VEL
LIN {X 0,Y 616.992,Z 344.373,A -85,B 0,C 180,E1 -6309.515,E2 -6309.515} C_VEL
LIN {X 0,Y 616.956,Z 344.377,A -85,B 0,C 180,E1 -6312.67,E2 -6312.67} C_VEL
LIN {X 0,Y 616.979,Z 344.368,A -85,B 0,C 180,E1 -6315.51,E2 -6315.51} C_VEL
LIN {X 0,Y 616.961,Z 344.377,A -85,B 0,C 180,E1 -6318.717,E2 -6318.717} C_VEL
LIN {X 0,Y 616.977,Z 344.362,A -85,B 0,C 180,E1 -6321.585,E2 -6321.585} C_VEL
LIN {X 0,Y 616.959,Z 344.363,A -85,B 0,C 180,E1 -6324.827,E2 -6324.827} C_VEL
LIN {X 0,Y 616.987,Z 344.374,A -85,B 0,C 180,E1 -6327.767,E2 -6327.767} C_VEL
LIN {X 0,Y 616.961,Z 344.379,A -85,B 0,C 180,E1 -6330.914,E2 -6330.914} C_VEL
LIN {X 0,Y 616.988,Z 344.363,A -85,B 0,C 180,E1 -6333.882,E2 -6333.882} C_VEL
LIN {X 0,Y 616.958,Z 344.372,A -85,B 0,C 180,E1 -6337.078,E2 -6337.078} C_VEL
LIN {X 0,Y 616.984,Z 344.368,A -85,B 0,C 180,E1 -6339.955,E2 -6339.955} C_VEL
LIN {X 0,Y 616.958,Z 344.354,A -85,B 0,C 180,E1 -6343.172,E2 -6343.172} C_VEL
LIN {X 0,Y 617.003,Z 344.371,A -85,B 0,C 180,E1 -6346.213,E2 -6346.213} C_VEL
LIN {X 0,Y 616.958,Z 344.381,A -85,B 0,C 180,E1 -6349.344,E2 -6349.344} C_VEL
LIN {X 0,Y 616.962,Z 344.424,A -85,B 0,C 180,E1 -6349.688,E2 -6349.688} C_VEL
LIN {X 0,Y 619.286,Z 350.473,A -85,B 0,C 180,E1 -6350.441,E2 -6350.441} C_VEL
LIN {X 0,Y 635.41,Z 376.25,A -85,B 0,C 180,E1 -6352.071,E2 -6352.071} C_VEL
LIN {X 0,Y 635.947,Z 377.186,A -85,B 0,C 180,E1 -6352.125,E2 -6352.125} C_VEL
LIN {X 0,Y 637.696,Z 381.876,A -85,B 0,C 180,E1 -6352.322,E2 -6352.322} C_VEL
LIN {X 0,Y 638.342,Z 388.319,A -85,B 0,C 180,E1 -6352.461,E2 -6352.461} C_VEL
LIN {X 0,Y 637.479,Z 398.608,A -85,B 0,C 180,E1 -6352.544,E2 -6352.544} C_VEL
LIN {X 0,Y 636.01,Z 411.557,A -85,B 0,C 180,E1 -6352.621,E2 -6352.621} C_VEL
LIN {X 0,Y 635.973,Z 412.733,A -85,B 0,C 180,E1 -6352.635,E2 -6352.635} C_VEL
LIN {X 0,Y 631.746,Z 660.219,A -85,B 0,C 180,E1 -6355.811,E2 -6355.811} C_VEL
LIN {X 0,Y 630.304,Z 739.834,A -85,B 0,C 180,E1 -6356.846,E2 -6356.846} C_VEL
LIN {X 0,Y 629.304,Z 764.933,A -85,B 0,C 180,E1 -6357.332,E2 -6357.332} C_VEL
LIN {X 0,Y 628.251,Z 784.817,A -85,B 0,C 180,E1 -6357.844,E2 -6357.844} C_VEL
LIN {X 0,Y 626.858,Z 807.75,A -85,B 0,C 180,E1 -6358.581,E2 -6358.581} C_VEL
LIN {X 0,Y 625.122,Z 830.21,A -85,B 0,C 180,E1 -6359.48,E2 -6359.48} C_VEL
LIN {X 0,Y 623.405,Z 851.74,A -85,B 0,C 180,E1 -6360.501,E2 -6360.501} C_VEL
LIN {X 0,Y 621.518,Z 872.423,A -85,B 0,C 180,E1 -6361.667,E2 -6361.667} C_VEL
LIN {X 0,Y 619.797,Z 890.524,A -85,B 0,C 180,E1 -6362.835,E2 -6362.835} C_VEL
LIN {X 0,Y 617.646,Z 912.113,A -85,B 0,C 180,E1 -6364.442,E2 -6364.442} C_VEL
LIN {X 0,Y 616.012,Z 928.638,A -85,B 0,C 180,E1 -6365.856,E2 -6365.856} C_VEL
LIN {X 0,Y 614.23,Z 946.758,A -85,B 0,C 180,E1 -6367.614,E2 -6367.614} C_VEL
LIN {X 0,Y 612.691,Z 963.333,A -85,B 0,C 180,E1 -6369.459,E2 -6369.459} C_VEL
LIN {X 0,Y 611.24,Z 980.108,A -85,B 0,C 180,E1 -6371.596,E2 -6371.596} C_VEL
LIN {X 0,Y 610.279,Z 992.662,A -85,B 0,C 180,E1 -6373.436,E2 -6373.436} C_VEL
LIN {X 0,Y 609.399,Z 1005.783,A -85,B 0,C 180,E1 -6375.655,E2 -6375.655} C_VEL
LIN {X 0,Y 608.841,Z 1015.497,A -85,B 0,C 180,E1 -6377.576,E2 -6377.576} C_VEL
LIN {X 0,Y 608.41,Z 1025.019,A -85,B 0,C 180,E1 -6379.776,E2 -6379.776} C_VEL
LIN {X 0,Y 608.139,Z 1032.381,A -85,B 0,C 180,E1 -6381.871,E2 -6381.871} C_VEL
LIN {X 0,Y 608.012,Z 1038.118,A -85,B 0,C 180,E1 -6383.864,E2 -6383.864} C_VEL
LIN {X 0,Y 607.934,Z 1043.234,A -85,B 0,C 180,E1 -6386.228,E2 -6386.228} C_VEL
LIN {X 0,Y 607.916,Z 1046.159,A -85,B 0,C 180,E1 -6388.209,E2 -6388.209} C_VEL
LIN {X 0,Y 607.901,Z 1048.057,A -85,B 0,C 180,E1 -6390.377,E2 -6390.377} C_VEL
LIN {X 0,Y 607.894,Z 1048.365,A -85,B 0,C 180,E1 -6392.64,E2 -6392.64} C_VEL
LIN {X 0,Y 607.899,Z 1047.404,A -85,B 0,C 180,E1 -6394.623,E2 -6394.623} C_VEL
LIN {X 0,Y 607.921,Z 1044.704,A -85,B 0,C 180,E1 -6396.991,E2 -6396.991} C_VEL
LIN {X 0,Y 607.97,Z 1040.79,A -85,B 0,C 180,E1 -6399.084,E2 -6399.084} C_VEL
LIN {X 0,Y 608.075,Z 1035.293,A -85,B 0,C 180,E1 -6401.284,E2 -6401.284} C_VEL
LIN {X 0,Y 608.286,Z 1028.026,A -85,B 0,C 180,E1 -6403.498,E2 -6403.498} C_VEL
LIN {X 0,Y 608.599,Z 1020.359,A -85,B 0,C 180,E1 -6405.436,E2 -6405.436} C_VEL
LIN {X 0,Y 609.176,Z 1009.276,A -85,B 0,C 180,E1 -6407.776,E2 -6407.776} C_VEL
LIN {X 0,Y 609.848,Z 998.896,A -85,B 0,C 180,E1 -6409.64,E2 -6409.64} C_VEL
LIN {X 0,Y 610.811,Z 985.692,A -85,B 0,C 180,E1 -6411.713,E2 -6411.713} C_VEL
LIN {X 0,Y 611.938,Z 971.742,A -85,B 0,C 180,E1 -6413.598,E2 -6413.598} C_VEL
LIN {X 0,Y 613.377,Z 955.934,A -85,B 0,C 180,E1 -6415.49,E2 -6415.49} C_VEL
LIN {X 0,Y 615.013,Z 938.663,A -85,B 0,C 180,E1 -6417.289,E2 -6417.289} C_VEL
LIN {X 0,Y 616.794,Z 921.137,A -85,B 0,C 180,E1 -6418.907,E2 -6418.907} C_VEL
LIN {X 0,Y 618.683,Z 901.859,A -85,B 0,C 180,E1 -6420.442,E2 -6420.442} C_VEL
LIN {X 0,Y 620.572,Z 882.575,A -85,B 0,C 180,E1 -6421.795,E2 -6421.795} C_VEL
LIN {X 0,Y 622.515,Z 861.552,A -85,B 0,C 180,E1 -6423.055,E2 -6423.055} C_VEL
LIN {X 0,Y 624.171,Z 842.465,A -85,B 0,C 180,E1 -6424.048,E2 -6424.048} C_VEL
LIN {X 0,Y 626.019,Z 819.2,A -85,B 0,C 180,E1 -6425.072,E2 -6425.072} C_VEL
LIN {X 0,Y 627.409,Z 798.552,A -85,B 0,C 180,E1 -6425.823,E2 -6425.823} C_VEL
LIN {X 0,Y 628.81,Z 774.942,A -85,B 0,C 180,E1 -6426.524,E2 -6426.524} C_VEL
LIN {X 0,Y 629.874,Z 751.394,A -85,B 0,C 180,E1 -6427.042,E2 -6427.042} C_VEL
LIN {X 0,Y 630.648,Z 727.106,A -85,B 0,C 180,E1 -6427.43,E2 -6427.43} C_VEL
LIN {X 0,Y 635.022,Z 474.062,A -85,B 0,C 180,E1 -6430.672,E2 -6430.672} C_VEL
LIN {X 0,Y 636.398,Z 391.316,A -85,B 0,C 180,E1 -6431.762,E2 -6431.762} C_VEL
LIN {X 0,Y 623.168,Z 369.368,A -85,B 0,C 180,E1 -6433.142,E2 -6433.142} C_VEL
LIN {X 0,Y 612.17,Z 352.556,A -85,B 0,C 180,E1 -6434.34,E2 -6434.34} C_VEL
LIN {X 0,Y 610.765,Z 350.187,A -85,B 0,C 180,E1 -6434.523,E2 -6434.523} C_VEL
LIN {X 0,Y 609.052,Z 345.365,A -85,B 0,C 180,E1 -6435.197,E2 -6435.197} C_VEL
LIN {X 0,Y 609.018,Z 345.347,A -85,B 0,C 180,E1 -6438.333,E2 -6438.333} C_VEL
LIN {X 0,Y 609.049,Z 345.361,A -85,B 0,C 180,E1 -6441.281,E2 -6441.281} C_VEL
LIN {X 0,Y 609.014,Z 345.33,A -85,B 0,C 180,E1 -6444.465,E2 -6444.465} C_VEL
LIN {X 0,Y 609.056,Z 345.365,A -85,B 0,C 180,E1 -6447.42,E2 -6447.42} C_VEL
LIN {X 0,Y 609.018,Z 345.364,A -85,B 0,C 180,E1 -6450.6,E2 -6450.6} C_VEL
LIN {X 0,Y 609.062,Z 345.365,A -85,B 0,C 180,E1 -6453.583,E2 -6453.583} C_VEL
LIN {X 0,Y 609.017,Z 345.365,A -85,B 0,C 180,E1 -6456.692,E2 -6456.692} C_VEL
LIN {X 0,Y 609.054,Z 345.361,A -85,B 0,C 180,E1 -6459.632,E2 -6459.632} C_VEL
LIN {X 0,Y 609.013,Z 345.36,A -85,B 0,C 180,E1 -6462.851,E2 -6462.851} C_VEL
LIN {X 0,Y 609.066,Z 345.353,A -85,B 0,C 180,E1 -6465.841,E2 -6465.841} C_VEL
LIN {X 0,Y 609.015,Z 345.363,A -85,B 0,C 180,E1 -6468.925,E2 -6468.925} C_VEL
LIN {X 0,Y 609.069,Z 345.365,A -85,B 0,C 180,E1 -6471.979,E2 -6471.979} C_VEL
LIN {X 0,Y 609.01,Z 345.359,A -85,B 0,C 180,E1 -6475.102,E2 -6475.102} C_VEL
LIN {X 0,Y 609.068,Z 345.352,A -85,B 0,C 180,E1 -6478.118,E2 -6478.118} C_VEL
LIN {X 0,Y 609.012,Z 345.365,A -85,B 0,C 180,E1 -6481.223,E2 -6481.223} C_VEL
LIN {X 0,Y 609.075,Z 345.361,A -85,B 0,C 180,E1 -6484.331,E2 -6484.331} C_VEL
LIN {X 0,Y 609.008,Z 345.352,A -85,B 0,C 180,E1 -6487.402,E2 -6487.402} C_VEL
LIN {X 0,Y 609.075,Z 345.351,A -85,B 0,C 180,E1 -6490.47,E2 -6490.47} C_VEL
LIN {X 0,Y 609.01,Z 345.366,A -85,B 0,C 180,E1 -6493.579,E2 -6493.579} C_VEL
LIN {X 0,Y 609.077,Z 345.357,A -85,B 0,C 180,E1 -6496.598,E2 -6496.598} C_VEL
LIN {X 0,Y 609.007,Z 345.352,A -85,B 0,C 180,E1 -6499.669,E2 -6499.669} C_VEL
LIN {X 0,Y 609.082,Z 345.35,A -85,B 0,C 180,E1 -6502.693,E2 -6502.693} C_VEL
LIN {X 0,Y 609.01,Z 345.366,A -85,B 0,C 180,E1 -6505.791,E2 -6505.791} C_VEL
LIN {X 0,Y 609.077,Z 345.361,A -85,B 0,C 180,E1 -6508.955,E2 -6508.955} C_VEL
LIN {X 0,Y 609.009,Z 345.367,A -85,B 0,C 180,E1 -6511.916,E2 -6511.916} C_VEL
LIN {X 0,Y 609.076,Z 345.363,A -85,B 0,C 180,E1 -6514.997,E2 -6514.997} C_VEL
LIN {X 0,Y 609.008,Z 345.366,A -85,B 0,C 180,E1 -6518.002,E2 -6518.002} C_VEL
LIN {X 0,Y 609.08,Z 345.362,A -85,B 0,C 180,E1 -6521.104,E2 -6521.104} C_VEL
LIN {X 0,Y 609.011,Z 345.369,A -85,B 0,C 180,E1 -6524.153,E2 -6524.153} C_VEL
LIN {X 0,Y 609.071,Z 345.565,A -85,B 0,C 180,E1 -6524.672,E2 -6524.672} C_VEL
LIN {X 0,Y 617.648,Z 366.692,A -85,B 0,C 180,E1 -6527.442,E2 -6527.442} C_VEL
LIN {X 0,Y 620.898,Z 374.872,A -85,B 0,C 180,E1 -6528.42,E2 -6528.42} C_VEL
LIN {X 0,Y 632.845,Z 395.363,A -85,B 0,C 180,E1 -6529.689,E2 -6529.689} C_VEL
LIN {X 0,Y 636.439,Z 411.894,A -85,B 0,C 180,E1 -6530.207,E2 -6530.207} C_VEL
LIN {X 0,Y 631.746,Z 678.208,A -85,B 0,C 180,E1 -6533.638,E2 -6533.638} C_VEL
LIN {X 0,Y 630.151,Z 767.053,A -85,B 0,C 180,E1 -6534.786,E2 -6534.786} C_VEL
LIN {X 0,Y 629.116,Z 792.394,A -85,B 0,C 180,E1 -6535.271,E2 -6535.271} C_VEL
LIN {X 0,Y 628.015,Z 812.716,A -85,B 0,C 180,E1 -6535.79,E2 -6535.79} C_VEL
LIN {X 0,Y 626.572,Z 836.174,A -85,B 0,C 180,E1 -6536.54,E2 -6536.54} C_VEL
LIN {X 0,Y 624.875,Z 858.359,A -85,B 0,C 180,E1 -6537.422,E2 -6537.422} C_VEL
LIN {X 0,Y 623.131,Z 880.429,A -85,B 0,C 180,E1 -6538.459,E2 -6538.459} C_VEL
LIN {X 0,Y 621.251,Z 901.593,A -85,B 0,C 180,E1 -6539.644,E2 -6539.644} C_VEL
LIN {X 0,Y 619.546,Z 920.145,A -85,B 0,C 180,E1 -6540.83,E2 -6540.83} C_VEL
LIN {X 0,Y 617.49,Z 941.596,A -85,B 0,C 180,E1 -6542.412,E2 -6542.412} C_VEL
LIN {X 0,Y 615.939,Z 958.032,A -85,B 0,C 180,E1 -6543.797,E2 -6543.797} C_VEL
LIN {X 0,Y 614.202,Z 976.677,A -85,B 0,C 180,E1 -6545.575,E2 -6545.575} C_VEL
LIN {X 0,Y 612.845,Z 991.46,A -85,B 0,C 180,E1 -6547.196,E2 -6547.196} C_VEL
LIN {X 0,Y 611.522,Z 1006.997,A -85,B 0,C 180,E1 -6549.118,E2 -6549.118} C_VEL
LIN {X 0,Y 610.387,Z 1021.24,A -85,B 0,C 180,E1 -6551.173,E2 -6551.173} C_VEL
LIN {X 0,Y 609.532,Z 1033.689,A -85,B 0,C 180,E1 -6553.219,E2 -6553.219} C_VEL
LIN {X 0,Y 608.878,Z 1044.639,A -85,B 0,C 180,E1 -6555.351,E2 -6555.351} C_VEL
LIN {X 0,Y 608.463,Z 1053.583,A -85,B 0,C 180,E1 -6557.376,E2 -6557.376} C_VEL
LIN {X 0,Y 608.158,Z 1061.907,A -85,B 0,C 180,E1 -6559.676,E2 -6559.676} C_VEL
LIN {X 0,Y 608.023,Z 1067.491,A -85,B 0,C 180,E1 -6561.584,E2 -6561.584} C_VEL
LIN {X 0,Y 607.945,Z 1072.696,A -85,B 0,C 180,E1 -6563.863,E2 -6563.863} C_VEL
LIN {X 0,Y 607.909,Z 1076.009,A -85,B 0,C 180,E1 -6566.039,E2 -6566.039} C_VEL
LIN {X 0,Y 607.906,Z 1077.836,A -85,B 0,C 180,E1 -6568.021,E2 -6568.021} C_VEL
LIN {X 0,Y 607.895,Z 1078.417,A -85,B 0,C 180,E1 -6570.377,E2 -6570.377} C_VEL
LIN {X 0,Y 607.908,Z 1077.495,A -85,B 0,C 180,E1 -6572.451,E2 -6572.451} C_VEL
LIN {X 0,Y 607.923,Z 1075.085,A -85,B 0,C 180,E1 -6574.717,E2 -6574.717} C_VEL
LIN {X 0,Y 607.957,Z 1071.102,A -85,B 0,C 180,E1 -6576.896,E2 -6576.896} C_VEL
LIN {X 0,Y 608.035,Z 1066.219,A -85,B 0,C 180,E1 -6578.892,E2 -6578.892} C_VEL
LIN {X 0,Y 608.266,Z 1058.66,A -85,B 0,C 180,E1 -6581.281,E2 -6581.281} C_VEL
LIN {X 0,Y 608.588,Z 1050.748,A -85,B 0,C 180,E1 -6583.298,E2 -6583.298} C_VEL
LIN {X 0,Y 609.123,Z 1040.402,A -85,B 0,C 180,E1 -6585.52,E2 -6585.52} C_VEL
LIN {X 0,Y 609.827,Z 1029.113,A -85,B 0,C 180,E1 -6587.559,E2 -6587.559} C_VEL
LIN {X 0,Y 610.779,Z 1016.117,A -85,B 0,C 180,E1 -6589.609,E2 -6589.609} C_VEL
LIN {X 0,Y 611.957,Z 1001.612,A -85,B 0,C 180,E1 -6591.57,E2 -6591.57} C_VEL
LIN {X 0,Y 613.372,Z 985.999,A -85,B 0,C 180,E1 -6593.438,E2 -6593.438} C_VEL
